// TwinCAT 3 PLC project ItemSimulator
// ProgramVersion: 3.1.4024.0
// libraries:
//   IO-Link Base, * (IO-Link)
//   SICK_IOL_Color, * (SICK AG)
//   Tc2_ModbusRTU, * (Beckhoff Automation GmbH)
//   Tc2_Standard, * (Beckhoff Automation GmbH)
//   Tc2_System, * (Beckhoff Automation GmbH)
//   Tc2_SystemCX, * (Beckhoff Automation GmbH)
//   Tc2_TcpIp, * (Beckhoff Automation GmbH)
//   Tc2_Utilities, * (Beckhoff Automation GmbH)
//   Tc3_Module, * (Beckhoff Automation GmbH)
//   TcUnit, * (www.tcunit.org)
//   VisuDialogs, * (System)
//   VisuSymbols,3.5.10.0,System
// project tree:
//   DUTs/ItemSimulator/ E_ItemGenerator.TcDUT, ST_ItemSimulator_HMI_CMD.TcDUT, ST_ItemSimulator_HMI_Status.TcDUT, ST_ItemSimulator_IO.TcDUT, ST_ItemGenerator.TcDUT
//   DUTs/TCP/ ST_TCPConnection.TcDUT, ST_TCPConnection_HMI_CMD.TcDUT, ST_TCPConnection_HMI_Status.TcDUT, ST_TCPConnection_IO.TcDUT
//   DUTs/TimeStamp/ ST_Timestamp_HMI_CMD.TcDUT, ST_Timestamp_HMI_Status.TcDUT, ST_Timestamp_IO.TcDUT
//   / GlobalTextList.TcGTLO, PlcTask.TcTTO, TCPTask.TcTTO, Visualization Manager.TcVMO (not stored)
//   GVLs/ GVL_Constant.TcGVL, GVL_HMI.TcGVL, GVL_IO.TcGVL
//   POUs/00_BuildingBlocks/ByteFunc/ FUN_GetHighByte.TcPOU, FUN_GetLowByte.TcPOU
//   POUs/00_BuildingBlocks/Calculation/ FB_FirstOrderLowPass.TcPOU, FUN_AngleCalculate.TcPOU, FUN_AngleChange.TcPOU, FUN_CartesianToPolar.TcPOU, FUN_Interpolation.TcPOU, FUN_LookUpTable.TcPOU, FUN_MinMaxSumAvg_6Reals.TcPOU, FUN_PolarToCartesian.TcPOU, FUN_Saturation.TcPOU, FUN_SaturationPointer.TcPOU, FUN_SaturationPointer_Int.TcPOU, FUN_SaturationPointer_UInt.TcPOU, FUN_Saturation_Int.TcPOU, FUN_Scale.TcPOU, ST_Coordinate.TcDUT
//   POUs/00_BuildingBlocks/Control/ FB_AliveCheck.TcPOU, FB_ClockPuls.TcPOU, FB_ClockPulsDetailed.TcPOU (not stored), FB_ClockPulsNumber.TcPOU, FB_EventHold.TcPOU, FB_FormatStringExtended.TcPOU, FB_Queue.TcPOU, FB_RampLimiter.TcPOU, FB_RangeSupervision.TcPOU, FB_SignalDead.TcPOU, FB_SteadyValue.TcPOU, FUN_InPos.TcPOU, FUN_InsideHysteresis.TcPOU, FUN_InsideHysteresis180pm.TcPOU, FUN_InsideHysteresis360.TcPOU, FUN_RangeInside.TcPOU, FUN_RangeOutside.TcPOU, FUN_GetHighLowValue.TcPOU
//   POUs/00_BuildingBlocks/Convert/ FUN_ConvFourByteToInt32.TcPOU, FUN_ConvFourByteToReal32.TcPOU, FUN_ConvFourByteToUdint32.TcPOU, FUN_ConvReal32ToFourByte.TcPOU, FUN_ConvTwoByteToInt16.TcPOU, FUN_ConvOneByteToUint8.TcPOU, FUN_ConvTwoByteToUInt16.TcPOU, U_Convert_INT16.TcDUT, U_Convert_UINT8.TcDUT, U_Convert_INT32.TcDUT, U_Convert_REAL32.TcDUT, U_Convert_UDINT32.TcDUT, U_Convert_UINT16.TcDUT, U_Convert_USINT.TcDUT
//   POUs/00_BuildingBlocks/EtherCAT/ FB_EK1101_Check.TcPOU, FB_HardwareCheck.TcPOU
//   POUs/00_BuildingBlocks/File/DUTs/ E_FileHandler_State.TcDUT
//   POUs/00_BuildingBlocks/File/ FB_FileHandler.TcPOU
//   POUs/00_BuildingBlocks/Modbus/DUTs/ E_ModbusRtuMaster_State.TcDUT, E_Modbus_DataType.TcDUT, ST_ModbusRtuMaster_StateLogEntry.TcDUT, ST_Modbus_Parameter.TcDUT, ST_Modbus_Unit.TcDUT
//   POUs/00_BuildingBlocks/Modbus/ FB_ModbusRtuMaster.TcPOU, FB_ModbusRtuMaster_20220719_1144.TcPOU, PRG_ModbusTest.TcPOU
//   POUs/00_BuildingBlocks/PlcToPlcCom/DUTs/ ADS_ErrorCodes.TcTLO, E_PlcAdsReadStep.TcDUT, ST_ComTest.TcDUT, ST_PlcAdsReadHmi.TcDUT
//   POUs/00_BuildingBlocks/PlcToPlcCom/ FB_PlcAdsRead.TcPOU, PRG_PlcAdsRead_Example.TcPOU, VIZU_PlcAdsRead.TcVIS
//   POUs/00_BuildingBlocks/StringFunctions/ FB_SeperateFileAndPathName.TcPOU, FUN_AddValuleToString.TcPOU, FUN_GetDateWithoutSeperator.TcPOU, FUN_GetDateWithUnderscore.TcPOU, FUN_GetDate.TcPOU, FUN_GetTimestamp.TcPOU, FUN_GetTimestampWithMs.TcPOU, FUN_GetTime.TcPOU, FUN_RealToString.TcPOU, FUN_ReplaceDotWithComma.TcPOU, F_Replace.TcPOU
//   POUs/01_TestUnit/ TEST.TcPOU (not stored)
//   POUs/01_TestUnit/TimeStampRegistry/ FB_TimestampRegistryTest.TcPOU
//   POUs/CSV_File/ PRG_CSVRead.TcPOU, PRG_CSVWrite.TcPOU (not stored)
//   POUs/IO_Link_Master/ FB_ColourSensor.TcPOU, FB_CMS.TcPOU, PRG_IO_Link_Master.TcPOU
//   POUs/Item_Simulator/FBs/ FB_ItemGenerator.TcPOU, FB_ItemRegister.TcPOU
//   POUs/Item_Simulator/ PRG_Simulator.TcPOU (not stored)
//   POUs/ MAIN.TcPOU, TCPCom.TcPOU
//   POUs/TCP_IP_Client/FBs/ FB_ReadTCP.TcPOU, FB_WriteTCP.TcPOU
//   POUs/TCP_IP_Client/ PRG_TCPIP.TcPOU
//   POUs/Timestamp_Registry/FBs/ FB_ReadTime.TcPOU (not stored), FB_SystemTime.TcPOU (not stored)
//   POUs/Timestamp_Registry/ PRG_TimestampRegistry.TcPOU
//   VISUs/ ItemSimulator.TcVIS, TimeStampOnItems.TcVIS
// real-time tasks:
//   TASK PlcTask: cycle T#10ms, priority 20, ADS port 350
//   TASK TCPTask: cycle T#2ms, priority 1, ADS port 351
// I/O:
//   DEVICE Device 5 (EtherCAT), AmsNetId 169.254.58.74.6.1
//     Box 1 (ICE11-8IOL-G60L-V1D) [ICE11-8IOL-G60L-V1D]
//       modules: Module 1 (IOL_I_32byte), Module 2 (IOL_I_32byte), Module 3 (IOL_I_16byte), Module 4 (IOL_I_16byte), Module 5 (IOL_I_16byte), Module 6 (IOL_I_16byte), Module 7 (IOL_I_16byte), Module 8 (IOL_I_16byte), Module 9 (STD_IN_1bit_Ch.B), Module 10 (STD_IN_1bit_Ch.B), Module 11 (STD_IN_1bit_Ch.B), Module 12 (STD_IN_1bit_Ch.B), Module 13 (STD_IN_1bit_Ch.B), Module 14 (STD_IN_1bit_Ch.B), Module 15 (STD_IN_1bit_Ch.B), Module 16 (STD_IN_1bit_Ch.B), Module 17 (TxPDO DI/IOL status), Module 18 (TxPDO New Diag Messages flag), Module 19 (TxPDO Timestamp), Module 20 (RxPDO DO/IOL control)
// variable links:
//   ItemSimulator/ItemSimulator Instance <-> Device 5 (EtherCAT)/Box 1 (ICE11-8IOL-G60L-V1D)
//     PlcTask Inputs/PRG_IO_Link_Master.fbCMS.arrCMSData <-> Module 2 (IOL_I_32byte)/TxPDO/input byte 0
//     PlcTask Inputs/PRG_IO_Link_Master.fbCMS.arrCMSData @bit {8..152 step 8} <-> Module 2 (IOL_I_32byte)/TxPDO/input byte {1..19}  (19 links)
//     PlcTask Inputs/PRG_IO_Link_Master.fbColorSensor.arrColorSensorData <-> Module 1 (IOL_I_32byte)/TxPDO/input byte 0
//     PlcTask Inputs/PRG_IO_Link_Master.fbColorSensor.arrColorSensorData @bit {8..88 step 8} <-> Module 1 (IOL_I_32byte)/TxPDO/input byte {1..11}  (11 links)
//     PlcTask Inputs/PRG_IO_Link_Master.fbColorSensor.nChannelStatus <-> IO-Link Port Status/Status of IO-Link Port 1

CONFIGURATION ItemSimulator
    RESOURCE PLC ON TwinCAT3
        TASK PlcTask(INTERVAL := T#10ms, PRIORITY := 20);
        TASK TCPTask(INTERVAL := T#2ms, PRIORITY := 1);
        PROGRAM MAIN WITH PlcTask : MAIN;
        PROGRAM TCPCom WITH TCPTask : TCPCom;
    END_RESOURCE
END_CONFIGURATION

// ---- DUTs/ItemSimulator/E_ItemGenerator.TcDUT
{attribute 'qualified_only'}
{attribute 'strict'}
TYPE E_ItemGenerator :
(
	Idle 						:= 0,
	ItemGenerator1 				:= 1,
	ItemGenerator2 				:= 2,
	ItemGenerator3 				:= 3,
	ItemGenerator4 				:= 4,
	ItemGenerator5 				:= 5,
	ItemGenerator6 				:= 6,
	ItemGenerator7 				:= 7,
	ItemGenerator8 				:= 8,
	ItemGenerator9 				:= 9,
	ItemGenerator10 			:= 10,
	ItemGeneratorFromRegistry	:= 11
	
);
END_TYPE

// ---- DUTs/ItemSimulator/ST_ItemSimulator_HMI_CMD.TcDUT
TYPE ST_ItemSimulator_HMI_CMD :
STRUCT
	bResetRegistry				:BOOL;
	bStartGenerator				:BOOL;
	bStopGenerator				:BOOL;
END_STRUCT
END_TYPE

// ---- DUTs/ItemSimulator/ST_ItemSimulator_HMI_Status.TcDUT
TYPE ST_ItemSimulator_HMI_Status :
STRUCT
END_STRUCT
END_TYPE

// ---- DUTs/ItemSimulator/ST_ItemSimulator_IO.TcDUT
TYPE ST_ItemSimulator_IO :
STRUCT
	bSignalOut	AT %Q* 			:BOOL;
	bSignalIn	AT %I* 			:BOOL;
END_STRUCT
END_TYPE

// ---- DUTs/ItemSimulator/ST_ItemGenerator.TcDUT
TYPE ST_ItemGenerator :
STRUCT
	bEnableGenerator		:BOOL;
	nNumberOfPulses			:UINT;
	tTimeOnPulse			:TIME;
	tTimeOffPulse			:TIME;
	bOutput					:BOOL;
END_STRUCT
END_TYPE

// ---- DUTs/TCP/ST_TCPConnection.TcDUT
TYPE ST_TCPConnection :
STRUCT
	bSocketConnect		:BOOL;
	sRemoteHost			:STRING;
	nRemotePort			:UDINT;
	tTimeOut			:TIME;
	bReset				:BOOL;
END_STRUCT
END_TYPE

// ---- DUTs/TCP/ST_TCPConnection_HMI_CMD.TcDUT
TYPE ST_TCPConnection_HMI_CMD :
STRUCT
	bWriteSocketConnect		:BOOL;
	bReadSocketConnect		:BOOL;
	bResetRegistry			:BOOL;
END_STRUCT
END_TYPE

// ---- DUTs/TCP/ST_TCPConnection_HMI_Status.TcDUT
TYPE ST_TCPConnection_HMI_Status :
STRUCT
	bCameraReadSocketIsConnected	:BOOL;
	bHlzWriteSocketIsConnected		:BOOL;
	
	aEANRegistry					:ARRAY[0..GVL_Constant.ITEM_ARRAY_SIZE] OF T_MaxString;
END_STRUCT
END_TYPE

// ---- DUTs/TCP/ST_TCPConnection_IO.TcDUT
TYPE ST_TCPConnection_IO :
STRUCT
END_STRUCT
END_TYPE

// ---- DUTs/TimeStamp/ST_Timestamp_HMI_CMD.TcDUT
TYPE ST_Timestamp_HMI_CMD :
STRUCT
	bResetRegistry				:BOOL;
END_STRUCT
END_TYPE

// ---- DUTs/TimeStamp/ST_Timestamp_HMI_Status.TcDUT
TYPE ST_Timestamp_HMI_Status :
STRUCT
	//Delta time in ms from Digital sensor to camera TCP
	aDeltaTimeMS			:ARRAY[0..GVL_Constant.ITEM_ARRAY_SIZE] OF UDINT;
	//Digital input sensor
	aDigitalSensorTime		:ARRAY[0..ITEM_ARRAY_SIZE] OF STRING;
	//Camera TCP port
	aTCPPortCameraTime		:ARRAY[0..ITEM_ARRAY_SIZE] OF STRING;
END_STRUCT
END_TYPE

// ---- DUTs/TimeStamp/ST_Timestamp_IO.TcDUT
TYPE ST_Timestamp_IO :
STRUCT
	bCameraOutSignal	AT %Q* 	:BOOL;
END_STRUCT
END_TYPE

// ---- POUs/00_BuildingBlocks/Calculation/ST_Coordinate.TcDUT
TYPE ST_Coordinate:
STRUCT
	rPosX			:LREAL;				// [mm] X-axis, Coordinate
	rPosY			:LREAL;				// [mm] Y-axis, Coordinate
	rPosTheta		:LREAL;				// [deg] Z-axis, Angle
END_STRUCT
END_TYPE

// ---- POUs/00_BuildingBlocks/Convert/U_Convert_INT16.TcDUT
TYPE U_Convert_INT16 :
UNION
	nValue		:INT;
	arrByte		:ARRAY[1..2] OF BYTE;
END_UNION
END_TYPE

// ---- POUs/00_BuildingBlocks/Convert/U_Convert_UINT8.TcDUT
TYPE U_Convert_UINT8 :
UNION
	nValue		:UINT;
	nBYTE		:BYTE;
END_UNION
END_TYPE

// ---- POUs/00_BuildingBlocks/Convert/U_Convert_INT32.TcDUT
TYPE U_Convert_INT32 :
UNION
	nValue		:DINT;
	arrByte		:ARRAY[1..4] OF BYTE;
END_UNION
END_TYPE

// ---- POUs/00_BuildingBlocks/Convert/U_Convert_REAL32.TcDUT
TYPE U_Convert_REAL32 :
UNION
	fValue		:REAL;
	arrByte		:ARRAY[1..4] OF BYTE;
END_UNION
END_TYPE

// ---- POUs/00_BuildingBlocks/Convert/U_Convert_UDINT32.TcDUT
TYPE U_Convert_UDINT32 :
UNION
	nValue		:UDINT;
	arrByte		:ARRAY[1..4] OF BYTE;
END_UNION
END_TYPE

// ---- POUs/00_BuildingBlocks/Convert/U_Convert_UINT16.TcDUT
TYPE U_Convert_UINT16 :
UNION
	nValue		:UINT;
	arrByte		:ARRAY[1..2] OF BYTE;
END_UNION
END_TYPE

// ---- POUs/00_BuildingBlocks/Convert/U_Convert_USINT.TcDUT
TYPE U_Convert_USINT :
UNION
	nValue		:USINT;					// Unsigned short integer value representation of data
    byValue 	:BYTE;					// Byte value representation of data
	//arrBit		:ARRAY[0..7]OF bool;	   // Bit representation of data
END_UNION
END_TYPE

// ---- POUs/00_BuildingBlocks/File/DUTs/E_FileHandler_State.TcDUT
{attribute 'qualified_only'}
{attribute 'strict'}
TYPE E_FileHandler_State :
(
	eReset				:= 0,
	eIdle				:= 10,
	
	eOpenFilePre		:= 20,
	eOpenFilePeri		:= 30,
	
	eReadFilePre		:= 40,
	eReadFilePeri		:= 50,

	eWriteFilePre		:= 60,
	eWriteFileSetLine	:= 65,
	eWriteFilePeri		:= 70,
	
	eCloseFilePre		:= 80,
	eCloseFilePeri		:= 90,

	eProcessFile		:= 100,
	
	eCopyFilePre		:= 200,
	eCopyFilePeri		:= 210,
	
	eDelFilePre			:= 220,
	eDelFilePeri		:= 230,
	
	eErrEntry			:= 900,
	eErrOpen			:= 910,
	eErrRead			:= 920,
	eErrWrite			:= 930,
	eErrClose			:= 940,
	eErrCopy			:= 950,
	eErrDel				:= 960
);
END_TYPE

// ---- POUs/00_BuildingBlocks/Modbus/DUTs/E_ModbusRtuMaster_State.TcDUT
{attribute 'qualified_only'}
{attribute 'strict'}
TYPE E_ModbusRtuMaster_State :
(
	eReset,
	eIdle,
	eReadPre,
	eReadPost,
	eError
);
END_TYPE

// ---- POUs/00_BuildingBlocks/Modbus/DUTs/E_Modbus_DataType.TcDUT
{attribute 'qualified_only'}
{attribute 'strict'}
TYPE E_Modbus_DataType :
(
	eInt16	 := 1,
	eInt32	 := 2
);
END_TYPE

// ---- POUs/00_BuildingBlocks/Modbus/DUTs/ST_ModbusRtuMaster_StateLogEntry.TcDUT
TYPE ST_ModbusRtuMaster_StateLogEntry :
STRUCT
	eStep				:E_ModbusRtuMaster_State;		// State
	sTimeEntry			:STRING;						// Timestamp for state entry
	iSecCount			:UDINT;							// Active time in state 	
END_STRUCT
END_TYPE

// ---- POUs/00_BuildingBlocks/Modbus/DUTs/ST_Modbus_Parameter.TcDUT
TYPE ST_Modbus_Parameter :
STRUCT
	nMemAddr			:WORD;
	nQuantity			:WORD;
	fConvFactor			:REAL;
	aDataStorage		:ARRAY[1..4] OF BYTE;
	aDataValue			:REAL;
	eDataType			:E_Modbus_DataType;
END_STRUCT
END_TYPE

// ---- POUs/00_BuildingBlocks/Modbus/DUTs/ST_Modbus_Unit.TcDUT
TYPE ST_Modbus_Unit :
STRUCT
	nAddr		:BYTE;
	aParam		:ARRAY[1..4] OF ST_Modbus_Parameter;		
END_STRUCT
END_TYPE

// ---- POUs/00_BuildingBlocks/PlcToPlcCom/DUTs/E_PlcAdsReadStep.TcDUT
//********************************************************************************
// E_PlcAdsReadStep
// ------------------------------------------------------------------------------- 
//
//	V2.00.00, HHL
// Baseline HST V1.01 10/4-16 (Valla V2.36)
//********************************************************************************
TYPE E_PlcAdsReadStep :
(
	eReset 				:= 0,		// Init
	eGetSymbolInfo 		:= 1,		// Get symbol infos
	eGetRemoteInfo 		:= 2,		// Get info (Index-Group/Offset)
	eWaitRemoteInfo 	:= 3,		// Wait for remote info
	eGetInfoError 		:= 4,		// Get info failed
	eIdle 				:= 10,		// Idle
	eRead 				:= 11,		// Read data
	eWaitReadDone 		:= 12,		// Wait read finished
	eWaitBeforeNextRead := 13, 		// Wait before next read
	eReadError 			:= 99		// Read failed
);
END_TYPE

// ---- POUs/00_BuildingBlocks/PlcToPlcCom/DUTs/ST_ComTest.TcDUT
TYPE ST_ComTest :
STRUCT
	bBool : BOOL;
	iInt : INT;
END_STRUCT
END_TYPE

// ---- POUs/00_BuildingBlocks/PlcToPlcCom/DUTs/ST_PlcAdsReadHmi.TcDUT
//********************************************************************************
// ST_PlcAdsReadHmi
// ------------------------------------------------------------------------------- 
//
//	V2.00.00, HHL
// Baseline HST V1.01 10/4-16 (Valla V2.36)
//********************************************************************************
TYPE ST_PlcAdsReadHmi :
STRUCT
	sRemoteId 				:STRING; 			// Remote NetId
	sRemoteSymbol 			:STRING;			// Remote variable
	bC_Init 				:BOOL; 				// Init request
	bS_Enable 				:BOOL; 				// Enable
	bS_LinkOk 				:BOOL; 				// Link to remote plc is ok
	bS_Error 				:BOOL; 				// Error
	eS_Step 				:E_PlcAdsReadStep;	// Step
	eS_ErrorStep		 	:E_PlcAdsReadStep;	// Error step
	udiS_ErrorId 			:UDINT; 			// Error id (ads)
	udiS_ReadCount 			:UDINT;  			// No of reads
	udiS_ReadErrors 		:UDINT; 			// No of read errors
	udiS_ReadIntervalErrors :UDINT;				// Read interval error
END_STRUCT
END_TYPE

// ---- GVLs/GVL_Constant.TcGVL
VAR_GLOBAL CONSTANT
	MAX_CSV_ROWS 			: UDINT := 100;
	MAX_CSV_COLUMNS 		: UDINT := 5;
	MAX_CSV_FIELD_LENGTH	: UDINT := 100;
	ITEM_ARRAY_SIZE			: INT:=10000;
END_VAR

// ---- GVLs/GVL_HMI.TcGVL
{attribute 'qualified_only'}
VAR_GLOBAL
	
	//Commands
	stItemSimulatorCmd		:ST_ItemSimulator_HMI_CMD;
	stTCPConnectionCmd		:ST_TCPConnection_HMI_CMD;
	stTimestampCmd			:ST_Timestamp_HMI_CMD;
	
	
	//Status
	stItemSimulatorStatus	:ST_ItemSimulator_HMI_Status;
	stTCPConnectionStatus	:ST_TCPConnection_HMI_Status;
	stTimestampStatus		:ST_Timestamp_HMI_Status;
END_VAR

// ---- GVLs/GVL_IO.TcGVL
{attribute 'qualified_only'}
VAR_GLOBAL
	stItemSimulator		:ST_ItemSimulator_IO;
	stTCPConnection		:ST_TCPConnection_IO;
	stTimestamp			:ST_Timestamp_IO;
END_VAR

// ---- POUs/MAIN.TcPOU
PROGRAM MAIN
VAR
END_VAR


//PRG_CSVRead();
//PRG_CSVWrite();

//Call Programs
PRG_Simulator();
PRG_TimestampRegistry();

PRG_IO_Link_Master();

END_PROGRAM

// ---- POUs/Timestamp_Registry/PRG_TimestampRegistry.TcPOU
PROGRAM PRG_TimestampRegistry
VAR 
	bInit					:BOOL := TRUE;
	fbReadTime				:FB_ReadTime;	
END_VAR

//Init
IF bInit THEN	
	bInit := FALSE;
END_IF

//Call read time
A_ReadTime();
	
//Reset Commands
GVL_HMI.stTimestampCmd.bResetRegistry := FALSE;

ACTION A_ReadTime:
fbReadTime(
	bReset := GVL_HMI.stTimestampCmd.bResetRegistry,
	bSignalIn := GVL_IO.stItemSimulator.bSignalIn,
	aDeltaTimeMS => GVL_HMI.stTimestampStatus.aDeltaTimeMS,
	aDigitalSensorTime => GVL_HMI.stTimestampStatus.aDigitalSensorTime,
	aTCPPortCameraTime => GVL_HMI.stTimestampStatus.aTCPPortCameraTime);
END_ACTION

END_PROGRAM

// ---- POUs/IO_Link_Master/PRG_IO_Link_Master.TcPOU
PROGRAM PRG_IO_Link_Master
VAR
	fbColorSensor			:FB_ColourSensor;
	fbCMS					:FB_CMS;
	
	bQL1					:BOOL; // Background
	bQL2					:BOOL; // Blue
	bQL3					:BOOL; // Green	
	bQL4					:BOOL; // None
	nQL1					:UINT;
	nQL2					:UINT;
	nQL3					:UINT;
	nQL4					:UINT;
	nValue					:INT;
	
	bEnable					:BOOL;
	bClear					:BOOL;
	arrColors				:ARRAY[0..GVL_Constant.ITEM_ARRAY_SIZE] OF INT;
	nI						:INT;
END_VAR

fbColorSensor(
	bQL1=>bQL1, 
	bQL2=>bQL2, 
	bQL3=>bQL3, 
	bQL4=>bQL4,
	nQL1=>nQL1,
	nQL2=>nQL2,
	nQL3=>nQL3,
	nQL4=>nQL4);
	
	
fbCMS();

nValue := fbColorSensor.nHighQLx;
IF NOT bQL1 AND NOT bClear THEN
	FOR nI := 0 TO GVL_Constant.ITEM_ARRAY_SIZE DO
		arrColors[nI] := fbColorSensor.nHighQLx;
	END_FOR
	
END_IF


IF bClear THEN
	FOR nI := 0 TO GVL_Constant.ITEM_ARRAY_SIZE DO
		arrColors[nI] := 0;
	END_FOR
END_IF

END_PROGRAM

// ---- POUs/IO_Link_Master/FB_ColourSensor.TcPOU
FUNCTION_BLOCK FB_ColourSensor
VAR_INPUT
END_VAR
VAR_OUTPUT
	nQL1					:UINT;
	nQL2					:UINT;
	nQL3					:UINT;
	nQL4					:UINT;
	
	bQL1					:BOOL;
	bQL2					:BOOL;
	bQL3					:BOOL;
	bQL4					:BOOL;
	
	nHighQLx				:INT;
END_VAR
VAR
	arrColorSensorData		AT %I*: ARRAY[0..11] OF BYTE;
	nChannelStatus			AT %I*: USINT;	
	
	arrQint					:ARRAY[1..24] OF BOOL;
	
	
	QoRAlarm				:BOOL;
	PDInvalid				:BOOL;
END_VAR

///////  index 120 value 0  ///////

// CMV QLx
nQL1 := FUN_ConvTwoByteToUInt16(nValue1 := arrColorSensorData[7], nValue2 := arrColorSensorData[6]); // CMV QL1
nQL2 := FUN_ConvTwoByteToUInt16(nValue1 := arrColorSensorData[5], nValue2 := arrColorSensorData[4]); // CMV QL2 
nQL3 := FUN_ConvTwoByteToUInt16(nValue1 := arrColorSensorData[3], nValue2 := arrColorSensorData[2]); // CMV QL3	
nQL4 := FUN_ConvTwoByteToUInt16(nValue1 := arrColorSensorData[1], nValue2 := arrColorSensorData[0]); // CMV QL4

IF bQL1 THEN
	nHighQLx := 1;
ELSIF bQL2 THEN
	nHighQLx := 2;
ELSIF bQL3 THEN
	nHighQLx := 3;
ELSIF bQL4 THEN
	nHighQLx := 4;
END_IF


// Qint 1 - 8
arrQint[1] := arrColorSensorData[10].0; //Not adjusted
arrQint[2] := arrColorSensorData[10].1; //Not adjusted
arrQint[3] := arrColorSensorData[10].2; //Not adjusted
arrQint[4] := arrColorSensorData[10].3; //Not adjusted
arrQint[5] := arrColorSensorData[10].4; //Not adjusted
arrQint[6] := arrColorSensorData[10].5; //Not adjusted
arrQint[7] := arrColorSensorData[10].6; //Not adjusted
arrQint[8] := arrColorSensorData[10].7; //Not adjusted

// Qint 9 - 16
arrQint[9] := arrColorSensorData[9].0; //Not adjusted
arrQint[10] := arrColorSensorData[9].1; //Not adjusted
arrQint[11] := arrColorSensorData[9].2; //Not adjusted
arrQint[12] := arrColorSensorData[9].3; //Not adjusted
arrQint[13] := arrColorSensorData[9].4; //Not adjusted
arrQint[14] := arrColorSensorData[9].5; //Not adjusted
arrQint[15] := arrColorSensorData[9].6; //Not adjusted
arrQint[16] := arrColorSensorData[9].7; //Not adjusted

// Qint 17 - 24
arrQint[17] := arrColorSensorData[8].0; //Not adjusted
arrQint[18] := arrColorSensorData[8].1; //Not adjusted
arrQint[19] := arrColorSensorData[8].2; //Not adjusted
arrQint[20] := arrColorSensorData[8].3; //Not adjusted
arrQint[21] := arrColorSensorData[8].4; //Not adjusted
arrQint[22] := arrColorSensorData[8].5; //Not adjusted
arrQint[23] := arrColorSensorData[8].6; //Not adjusted
arrQint[24] := arrColorSensorData[8].7; //Not adjusted

//Alarms
QoRAlarm := arrColorSensorData[11].4;
PDInvalid := arrColorSensorData[11].5;

//Digital outputs
bQL1 := arrColorSensorData[11].0;
bQL2 := arrColorSensorData[11].1;
bQL3 := arrColorSensorData[11].2;
bQL4 := arrColorSensorData[11].3;

END_FUNCTION_BLOCK

// ---- POUs/00_BuildingBlocks/Convert/FUN_ConvTwoByteToUInt16.TcPOU
FUNCTION FUN_ConvTwoByteToUInt16 : UINT
VAR_INPUT
	nValue1		:BYTE;				// Input Byte no 1
	nValue2		:BYTE;				// Input Byte no 2
END_VAR
VAR
	uData		:U_Convert_UINT16;		// Data variable used for conversion
END_VAR


// Save input bytes in data union
uData.arrByte[1] := nValue1;
uData.arrByte[2] := nValue2;

// Return value
FUN_ConvTwoByteToUInt16 := uData.nValue;

END_FUNCTION

// ---- POUs/IO_Link_Master/FB_CMS.TcPOU
FUNCTION_BLOCK FB_CMS
VAR_INPUT
END_VAR
VAR_OUTPUT
	Impulse_X				:REAL;
	Impulse_Y				:REAL;
	Impulse_Z				:REAL;
	Temperature				:REAL;
END_VAR
VAR
	arrCMSData				AT %I*: ARRAY[0..19] OF BYTE;
	nChannelStatus			AT %I*: USINT;	
	
	AlarmTemperature		:BOOL;
	AlarmShock				:BOOL;
	AlarmRMS_PreMax			:BOOL;
	AlarmRMS_Max			:BOOL;
	
	ConfByte				:ARRAY[0..1] OF BYTE;
END_VAR


Impulse_X := FUN_ConvFourByteToReal32(nValue1 := arrCMSData[15], nValue2 := arrCMSData[14], nValue3 := arrCMSData[13], nValue4 := arrCMSData[12]); 
Impulse_Y := FUN_ConvFourByteToReal32(nValue1 := arrCMSData[11], nValue2 := arrCMSData[10], nValue3 := arrCMSData[9], nValue4 := arrCMSData[8]); 
Impulse_Z := FUN_ConvFourByteToReal32(nValue1 := arrCMSData[7], nValue2 := arrCMSData[6], nValue3 := arrCMSData[5], nValue4 := arrCMSData[4]); 
Temperature := FUN_ConvFourByteToReal32(nValue1 := arrCMSData[3], nValue2 := arrCMSData[2], nValue3 := arrCMSData[1], nValue4 := arrCMSData[0]); 



// Byte 18 - 19 is configureable byte. These can be set in SOPAS software.
ConfByte[0].0 := arrCMSData[18].0; // Deactivated
ConfByte[0].1 := arrCMSData[18].1; // Deactivated
ConfByte[0].2 := arrCMSData[18].2; // Deactivated
ConfByte[0].3 := arrCMSData[18].3; // Deactivated
ConfByte[0].4 := arrCMSData[18].4; // Deactivated
ConfByte[0].5 := arrCMSData[18].5; // Deactivated
ConfByte[0].6 := arrCMSData[18].6; // Deactivated
ConfByte[0].7 := arrCMSData[18].7; // Deactivated

ConfByte[1].0 := arrCMSData[19].0; // Deactivated
ConfByte[1].1 := arrCMSData[19].1; // Deactivated
ConfByte[1].2 := arrCMSData[19].2; // Deactivated
ConfByte[1].3 := arrCMSData[19].3; // Deactivated

AlarmTemperature := arrCMSData[19].4; 
AlarmShock := arrCMSData[19].5; 
AlarmRMS_PreMax := arrCMSData[19].6; 
AlarmRMS_Max := arrCMSData[19].7;

END_FUNCTION_BLOCK

// ---- POUs/00_BuildingBlocks/Convert/FUN_ConvFourByteToReal32.TcPOU
FUNCTION FUN_ConvFourByteToReal32 : REAL
VAR_INPUT
	nValue1		:BYTE;				// Input Byte no 1
	nValue2		:BYTE;				// Input Byte no 2
	nValue3		:BYTE;				// Input Byte no 3
	nValue4		:BYTE;				// Input Byte no 4
END_VAR
VAR
	uData		:U_Convert_REAL32;	// Data variable used for conversion
END_VAR


// Save input bytes in data union
uData.arrByte[1] := nValue1;
uData.arrByte[2] := nValue2;
uData.arrByte[3] := nValue3;
uData.arrByte[4] := nValue4;

// Return value
FUN_ConvFourByteToReal32 := uData.fValue;

END_FUNCTION

// ---- POUs/TCPCom.TcPOU
PROGRAM TCPCom
VAR
END_VAR

//Call programs
PRG_TCPIP();

END_PROGRAM

// ---- POUs/TCP_IP_Client/PRG_TCPIP.TcPOU
PROGRAM PRG_TCPIP 
VAR	
	bInit 						:BOOL := TRUE;
	bReset						:BOOL;
	
	stReadTCP					:ST_TCPConnection;
	fbReadFromCameraTCP			:FB_ReadTCP;
	bConnectToReadSocket		:BOOL;
	
	stWriteTCP					:ST_TCPConnection;
	fbWriteToHLZ				:FB_WriteTCP;
	bConnectToWriteSocket		:BOOL;
END_VAR

//Init
IF bInit THEN	
	bInit := FALSE;
END_IF


A_ReadFromCamera();
A_WriteToHlz();


//Reset Commands
GVL_HMI.stTCPConnectionCmd.bResetRegistry := FALSE;


IF GVL_HMI.stTCPConnectionCmd.bWriteSocketConnect THEN
	GVL_HMI.stTCPConnectionCmd.bReadSocketConnect := FALSE;
	
ELSIF GVL_HMI.stTCPConnectionCmd.bReadSocketConnect THEN
	GVL_HMI.stTCPConnectionCmd.bWriteSocketConnect := FALSE;
END_IF;

ACTION A_ReadFromCamera:
//Initialize Read TCP
stReadTCP.sRemoteHost := '10.12.5.10';
stReadTCP.nRemotePort := 51236;
stReadTCP.tTimeOut := T#45S;
stReadTCP.bSocketConnect := GVL_HMI.stTCPConnectionCmd.bReadSocketConnect;
stReadTCP.bReset := GVL_HMI.stTCPConnectionCmd.bResetRegistry;

//Call Read TCP
fbReadFromCameraTCP(
	stTCPConnection:=stReadTCP,
	aEANRegistry=>GVL_HMI.stTCPConnectionStatus.aEANRegistry,
	bIsConnected=>GVL_HMI.stTCPConnectionStatus.bCameraReadSocketIsConnected);
END_ACTION

ACTION A_WriteToHlz:
//Initialize Write TCP
stWriteTCP.sRemoteHost := '10.12.5.10';
stWriteTCP.nRemotePort := 51237;
stWriteTCP.tTimeOut := T#45S;
stWriteTCP.bSocketConnect := GVL_HMI.stTCPConnectionCmd.bWriteSocketConnect;
stWriteTCP.bReset := GVL_HMI.stTCPConnectionCmd.bResetRegistry;


//Call Write TCP
fbWriteToHLZ(
	aEANRegistry:=fbReadFromCameraTCP.aEANRegistry,
	stTCPConnection:=stWriteTCP,
	bIsConnected=>GVL_HMI.stTCPConnectionStatus.bHlzWriteSocketIsConnected);
END_ACTION

END_PROGRAM

// ---- POUs/TCP_IP_Client/FBs/FB_ReadTCP.TcPOU
FUNCTION_BLOCK FB_ReadTCP 
VAR_INPUT
	stTCPConnection		:ST_TCPConnection;
END_VAR
VAR_OUTPUT
	aEANRegistry		:ARRAY[0..GVL_Constant.ITEM_ARRAY_SIZE] OF T_MaxString;
	bIsConnected		:BOOL;
END_VAR
VAR_IN_OUT
END_VAR
VAR
	fbConnectSocket		:FB_SocketConnect;
	fbDisconnect		:FB_SocketClose;
	rConnectedSocket	:F_TRIG;
	tRefreshRead		:FB_ClockPulsDetailed;
	fbSocketRecive		:FB_SocketReceive;
	rReadComplete		:R_TRIG;
	aReadBytes			:ARRAY[0..1023] OF BYTE;
	sReadString			:T_MaxString;
	iRead				:UINT;
	i					:INT;

	bReadComplete		:BOOL;
	bResetEANRegistry	:BOOL;
	hSocket				:T_HSOCKET;
END_VAR


A_ConnectToReadSocket();

IF bIsConnected THEN
	A_ReadFromTCPSocket();
END_IF

ACTION A_ConnectToReadSocket:
IF stTCPConnection.bSocketConnect THEN

	//Connect read port
	fbConnectSocket(
		sRemoteHost:=stTCPConnection.sRemoteHost,
		nRemotePort:=stTCPConnection.nRemotePort, 
		bExecute:=TRUE,
		tTimeout:=stTCPConnection.tTimeOut,
		hSocket=>hSocket);
	ELSE
		//Disconnect read port
		fbConnectSocket(bExecute:=FALSE);
		fbDisconnect(hSocket:=hSocket);
		bIsConnected := FALSE;
END_IF

rConnectedSocket(CLK:=fbConnectSocket.bBusy);

IF rConnectedSocket.Q AND NOT fbConnectSocket.bError THEN
	bIsConnected := TRUE;
END_IF
END_ACTION

ACTION A_ReadFromTCPSocket:
IF bIsConnected THEN

	//Refresh read timer
	tRefreshRead(bEnable:=TRUE, tPulsLengthOn:=T#2MS, tPulsLengthOff:=T#2MS);
	
	fbSocketRecive(
		hSocket:=hSocket, 
		cbLen:=SIZEOF(aReadBytes),
		pDest:=ADR(aReadBytes),
		bExecute:=tRefreshRead.bPuls);
		
	rReadComplete(CLK:=fbSocketRecive.nRecBytes > 0);
	
	
	//If byte read, copy into string.
	IF rReadComplete.Q THEN
		MEMCPY(destAddr:=ADR(sReadString), srcAddr:=ADR(aReadBytes),n:=fbSocketRecive.nRecBytes);
		aEANRegistry[iRead] := sReadString;
		MEMSET(destAddr:=ADR(aReadBytes),fillByte:=0, n:=fbSocketRecive.nRecBytes);
		MEMSET(destAddr:=ADR(sReadString),fillByte:=0, n:=fbSocketRecive.nRecBytes);
		iRead:=iRead+1;
		bReadComplete:=TRUE;
	ELSE
		bReadComplete:=FALSE;
	END_IF
END_IF


//Reset registry of EAN strings
IF PRG_Simulator.bStartGenerator OR PRG_Simulator.bStopGenerator OR (PRG_Simulator.i > PRG_Simulator.nTimeCount) OR stTCPConnection.bReset THEN
	FOR i := 0 TO GVL_Constant.ITEM_ARRAY_SIZE DO 
		aEANRegistry[i] := '';
	END_FOR

	iRead := 0;
	MEMSET(destAddr:=ADR(aReadBytes),fillByte:=0, n:=fbSocketRecive.nRecBytes);
	MEMSET(destAddr:=ADR(sReadString),fillByte:=0, n:=fbSocketRecive.nRecBytes);	
	
	
	//Reset commands
	stTCPConnection.bReset :=FALSE;
END_IF
END_ACTION

END_FUNCTION_BLOCK

// ---- POUs/TCP_IP_Client/FBs/FB_WriteTCP.TcPOU
FUNCTION_BLOCK FB_WriteTCP 
VAR_INPUT
	stTCPConnection		:ST_TCPConnection;
	aEANRegistry		:ARRAY[0..GVL_Constant.ITEM_ARRAY_SIZE] OF T_MaxString;
END_VAR
VAR_OUTPUT
	bIsConnected		:BOOL;
END_VAR
VAR
	fbConnectSocket		:FB_SocketConnect;
	fbDisconnect		:FB_SocketClose;
	rConnectedSocket	:F_TRIG;
	fbSocketSend		:FB_SocketSend;
	rWriteComplete		:R_TRIG;
	aWriteBytes			:ARRAY[0..1023] OF BYTE;
	iWrite				:UINT;
	WriteSignal			:F_TRIG;
	nWriteLen			:UDINT;
	i					:INT;

	bWriteComplete		:BOOL;
	bResetEANRegistry	:BOOL;
	hSocket				:T_HSOCKET;
END_VAR


A_ConnectToWriteSocket();

IF bIsConnected THEN
	A_WriteToTCPSocket();
END_IF

ACTION A_ConnectToWriteSocket:
IF stTCPConnection.bSocketConnect THEN
	
	//Connect write port
	fbConnectSocket(
		sRemoteHost:=stTCPConnection.sRemoteHost,
		nRemotePort:=stTCPConnection.nRemotePort, 
		bExecute:=TRUE,
		tTimeout:=stTCPConnection.tTimeOut,
		hSocket=>hSocket);
	ELSE
		//Disconnect write port
		fbConnectSocket(bExecute:=FALSE);
		fbDisconnect(hSocket:=hSocket);
		bIsConnected := FALSE;
END_IF



rConnectedSocket(CLK:=fbConnectSocket.bBusy);

IF rConnectedSocket.Q AND NOT fbConnectSocket.bError THEN
	bIsConnected := TRUE;
END_IF
END_ACTION

ACTION A_WriteToTCPSocket:
IF bIsConnected THEN	
	//Falling edge of item generator
	WriteSignal(CLK:=GVL_IO.stItemSimulator.bSignalOut);
	
	IF WriteSignal.Q THEN
		//Get length of string written
		nWriteLen := INT_TO_UDINT(LEN(STR:=aEANRegistry[iWrite]));
	
		//Copy string into array of bytes
		MEMCPY(destAddr:=ADR(aWriteBytes),srcAddr:=ADR(aEANRegistry[iWrite]),n:=nWriteLen);
		iWrite := iWrite + 1;
	END_IF
		
	//Write byte array to TCP server
	fbSocketSend(
		hSocket:=hSocket, 
		cbLen:=nWriteLen,
		pSrc:=ADR(aWriteBytes),
		bExecute:=WriteSignal.Q AND PRG_Simulator.fbItemGenerator.stItemGenFromReg.bEnableGenerator);
END_IF;


//Reset registry of EAN strings
IF PRG_Simulator.bStartGenerator OR PRG_Simulator.bStopGenerator OR (PRG_Simulator.i > PRG_Simulator.nTimeCount) OR bResetEANRegistry THEN
	FOR i := 0 TO GVL_Constant.ITEM_ARRAY_SIZE DO 
		aEANRegistry[i] := '';
	END_FOR

	iWrite := 0;	
	
	//Reset Command
	bResetEANRegistry := FALSE;
END_IF
END_ACTION

END_FUNCTION_BLOCK

// ---- POUs/00_BuildingBlocks/ByteFunc/FUN_GetHighByte.TcPOU
FUNCTION FUN_GetHighByte : BYTE
VAR_INPUT
	wIn			:WORD;			
END_VAR
VAR
	byHigh		:BYTE;
END_VAR


// Get the high byte value from the word
byHigh.0 := wIn.8;
byHigh.1 := wIn.9;
byHigh.2 := wIn.10;
byHigh.3 := wIn.11;
byHigh.4 := wIn.12;
byHigh.5 := wIn.13;
byHigh.6 := wIn.14;
byHigh.7 := wIn.15;

// Return value
FUN_GetHighByte := byHigh;

END_FUNCTION

// ---- POUs/00_BuildingBlocks/ByteFunc/FUN_GetLowByte.TcPOU
FUNCTION FUN_GetLowByte : BYTE
VAR_INPUT
	wIn			:WORD;			
END_VAR
VAR
	byLow		:BYTE;
END_VAR


// Get the high byte value from the word
byLow.0 := wIn.0;
byLow.1 := wIn.1;
byLow.2 := wIn.2;
byLow.3 := wIn.3;
byLow.4 := wIn.4;
byLow.5 := wIn.5;
byLow.6 := wIn.6;
byLow.7 := wIn.7;

// Return value
FUN_GetLowByte := byLow;

END_FUNCTION

// ---- POUs/00_BuildingBlocks/Calculation/FB_FirstOrderLowPass.TcPOU
//********************************************************************************
// FB_FirstOrderLowPass.
// -------------------------------------------------------------------------------
// This FB implements a first order low pass filter after the equation:
// 					Y[n] = Alpha x Y[n-1]  +  Beta X[n]
// The FB must be called in every scan when used. Input values for frequency and
// cut-off frequency can be changed during filtration without reset of the filtered
// output value.
//
// Version:
//			- V1.00.00	HHL, 26/11-2019
//********************************************************************************
FUNCTION_BLOCK FB_FirstOrderLowPass
VAR_INPUT
	rSampleFrequency	:REAL;			// Sample time for algorithm in Hz
	rCutOffFrequency	:REAL;			// Cut off frequency for filter in Hz 	
	rXn					:REAL;			// Input value before filtration
	bReset				:BOOL;			// Filter memory is reset on a rising edge. Output is reset to zero
END_VAR

VAR_OUTPUT
	rYn					:REAL;			// Output value after filtration
END_VAR

VAR
	osReset				:R_TRIG;		// One shot for reset of filter
	rFrequencyRatio		:REAL;			// Frequency ration for determination of Beta value
	rAlpha				:REAL;			// Alpha value for first order filter
	rBeta				:REAL;			// Beta value for first order filter
	rSampleFrequencyOld	:REAL;			// Input setting from previous scan for sample time for algorithm in Hz
	rCutOffFrequencyOld	:REAL;			// Input setting from previous scan for cut off frequency for filter in Hz 
END_VAR

// Check if filter has been reset
osReset(CLK:= bReset, Q=> );

// Check if settings have chaged
IF (rSampleFrequency <> rSampleFrequencyOld) OR (rCutOffFrequency <> rCutOffFrequencyOld) OR osReset.Q THEN
	// Settings have changed => Calculate Alpha and Beta again
	rFrequencyRatio := rSampleFrequency/rCutOffFrequency;
	rBeta := LREAL_TO_REAL(1/(2*PI*rFrequencyRatio));
	rAlpha := 1 - rBeta;
	
	// Update "old" values
	rSampleFrequencyOld := rSampleFrequency;
	rCutOffFrequencyOld := rCutOffFrequency;
	
	// If reset was activated, then reset output value
	IF osReset.Q THEN
		rYn := 0;
	END_IF
END_IF

// Calculate filtered value
rYn := rAlpha*rYn + rBeta*rXn;

END_FUNCTION_BLOCK

// ---- POUs/00_BuildingBlocks/Calculation/FUN_AngleCalculate.TcPOU
//********************************************************************************
// FUN_AngleCalculate.
// -------------------------------------------------------------------------------
// This function calculates the angle between two coordinate points.
// Angle when moving from stCoor1 to stCoor2 (Exit angle for stCoor1, Entry angle for stCoor2) 
// The output angle is defined as plus/minus 180 degrees. 
//	
// Version:
//			- V1.00.00	HHL, 26/11-2019
//********************************************************************************
FUNCTION FUN_AngleCalculate : LREAL
VAR_IN_OUT
END_VAR
VAR_INPUT
	stCoor1			:ST_Coordinate;			// Coordinates from previous motion command line (If known)
	stCoor2			:ST_Coordinate;			// Coordinates from active line
END_VAR
VAR
	rTheta			:LREAL;					// [pm 180 deg] Angle when moving from stCoor1 to stCoor2 (Exit angle for stCoor1, Entry angle for stCoor2) 
	bError			:BOOL;					// True if error occured during determination of angle
	rX_Leg			:LREAL;					// Displacement in x-axis between x-pos from stCoor1 and stCoor2
	rY_Leg			:LREAL;					// Displacement in y-axis between y-pos from stCoor1 and stCoor2
END_VAR

// Angle (Theta) must be calculated from two positions. 
// Calculate the two "legs" formed by the triangle of postion from stCoor1 and stCoor2 
rX_Leg := stCoor2.rPosX - stCoor1.rPosX;
rY_Leg := stCoor2.rPosY - stCoor1.rPosY;

// Calculate angle "Theta"
IF rX_Leg = 0 OR rY_Leg = 0 THEN
	// Theta is a parallel line to either x-axis or y-axis
	IF rX_Leg = 0 AND rY_Leg > 0 THEN
		// Theta is parallel to positive direction on y-axis
		rTheta := 90.0;
	ELSIF rX_Leg = 0 AND rY_Leg < 0 THEN
		// Theta is parallel to negative direction on y-axis
		rTheta := -90.0;
	ELSIF rX_Leg > 0 AND rY_Leg = 0 THEN
		// Theta is parallel to positive direction on x-axis
		rTheta := 0.0;
	ELSIF rX_Leg < 0 AND rY_Leg = 0 THEN
		// Theta is parallel to negative direction on x-axis
		rTheta := 180.0;
	ELSIF rX_Leg = 0 AND rY_Leg = 0 THEN
		// Special case where both stCoor1 and stCoor2 have the same coordinates (Should not happen).
		bError := TRUE;
	END_IF	
ELSE
	// Calculate angle "Theta" from position in stCoor1 and stCoor2	 
	IF stCoor1.rPosX <= stCoor2.rPosX AND stCoor1.rPosY <= stCoor2.rPosY THEN
		// I. Quadrant	
		// Location of stCoor2 in regards to stCoor1 as center
		IF rX_Leg <> 0 THEN
			rTheta := RAD_TO_DEG(ATAN(rY_Leg/rX_Leg));
		ELSIF rX_Leg = 0 THEN
			IF rY_Leg > 0 THEN
				rTheta := 90.0;
			ELSIF rY_Leg = 0 THEN
				// Special case where both stCoor1 and stCoor2 have the same coordinates (Should not happen).
				bError := TRUE;
			END_IF
		END_IF
	ELSIF stCoor1.rPosX > stCoor2.rPosX AND stCoor1.rPosY <= stCoor2.rPosY THEN 	
		// II. Quadrant	
		// Location of stCoor2 in regards to stCoor1 as centers
		IF rY_Leg <> 0 THEN
			rTheta := RAD_TO_DEG(ATAN(rY_Leg/rX_Leg)) + 180;
		ELSIF rY_Leg = 0 THEN
			IF rX_Leg > 0 THEN
				rTheta := 0.0;
			ELSE
				rTheta := -180.0;
			END_IF
		END_IF
	ELSIF stCoor1.rPosX > stCoor2.rPosX AND stCoor1.rPosY > stCoor2.rPosY THEN 	
		// III. Quadrant	
		// Location of stCoor2 in regards to stCoor1 as center
		rTheta := -1*(180 - RAD_TO_DEG(ATAN(rY_Leg/rX_Leg)));
	ELSIF stCoor1.rPosX < stCoor2.rPosX AND stCoor1.rPosY > stCoor2.rPosY THEN 	
		// IV. Quadrant	
		// Location of stCoor2 in regards to stCoor1 as center
		rTheta := RAD_TO_DEG(ATAN(rY_Leg/rX_Leg));
	END_IF	
END_IF

// Return result
IF NOT bError THEN
	// No error => Return result.
	FUN_AngleCalculate := rTheta;
ELSE
	// Error => Return error value
	FUN_AngleCalculate := -999.0;
END_IF

END_FUNCTION

// ---- POUs/00_BuildingBlocks/Calculation/FUN_AngleChange.TcPOU
//********************************************************************************
// FUN_AngleChange.
// -------------------------------------------------------------------------------
// This function calculates the difference between to angles in degrees. Input and
// output values are all defined as plus/minus 180 degrees. 
//	
// Version:
//			- V1.00.00	HHL, 26/11-2019
//********************************************************************************
FUNCTION FUN_AngleChange : LREAL
VAR_INPUT
	rTheta1			:LREAL;			// [pm 180 deg] Theta angle from coordinate set 1
	rTheta2			:LREAL;			// [pm 180 deg] Theta angle from coordinate set 2
END_VAR
VAR
	rThetaChange	:LREAL;			// Change in angle between two points	
END_VAR

// Calculate change in theta angle
IF rTheta1 >= 0 AND rTheta2 >= 0 THEN
	// Both coordinates have a positive theta angle
	rThetaChange := rTheta2 - rTheta1;
ELSIF rTheta1 <= 0 AND rTheta2 <= 0 THEN
	// Both coordinates have a negative thata angle
	rThetaChange := rTheta2 - rTheta1;
ELSE
	// One coordinate set has a positive theta angle and the other has a negative
	IF rTheta1 >= 0 THEN
		// Coordinate set one has a positive coordinate set and coordinate 2 has a negative
		// First find angle when passing through 0 deg.
		rThetaChange := rTheta2 - rTheta1;
		IF ABS(rThetaChange) > 180 THEN
			// Angle is greather than 180 deg. Do not use angle that passes through 0 deg. 
			// Calculate the angle when passing through p/m 180 deg
			rThetaChange := 360 - ABS(rThetaChange);
		END_IF
	ELSE
		// Coordinate set one has a negative coordinate set and coordinate 2 has a positive
		// First find angle when passing through 0 deg.
		rThetaChange := rTheta2 - rTheta1;
		IF ABS(rThetaChange) > 180 THEN
			// Angle is greather than 180 deg. Do not use angle that passes through 0 deg. 
			// Calculate the angle when passing through p/m 180 deg
			rThetaChange := -1 * (360 - ABS(rThetaChange));
		END_IF
	END_IF
END_IF 

// Return result
FUN_AngleChange := rThetaChange;

END_FUNCTION

// ---- POUs/00_BuildingBlocks/Calculation/FUN_CartesianToPolar.TcPOU
//********************************************************************************
// FUN_Cartesian to polar.
// -------------------------------------------------------------------------------
// This function calculates the polar coordinates r and theta from
// the cartesian X and Y coordinates. 
//	
// Version:
//			- V1.01	HHL, 11/05-2022
//********************************************************************************
FUNCTION FUN_CartesianToPolar : LREAL
VAR_IN_OUT
END_VAR
VAR_INPUT
	fX				:REAL;			// X-axis coordinate
	fY				:REAL;			// Y-axis coordinate
END_VAR
VAR_OUTPUT
	fRadius			:REAL;			// Radius for polar coordinate
	fAngle			:REAL;			// [deg] Angle for polar coordinate 
END_VAR
VAR
	bError			:BOOL;			// True if error occured during determination of angle
END_VAR


// Calculate polar coordinates from cartesian coordinates
//-----------------------------------------

// Calculate radius
fRadius := LREAL_TO_REAL(SQRT((EXPT(fX,2) + EXPT(fY,2))));

// Calculate angle
IF fX <> 0 THEN 
	// Calculate angle 
	IF 0 <= fX AND 0 <= fY THEN
		// I. Quadrant	
		IF fX <> 0 THEN
			fAngle := LREAL_TO_REAL(RAD_TO_DEG(ATAN(fY/fX)));
		ELSIF fX = 0 THEN
			IF fY > 0 THEN
				fAngle := 90.0;
			ELSIF fY = 0 THEN
				// Special case where both fX and fY are zero.
				bError := TRUE;
			END_IF
		END_IF
	ELSIF 0 > fX AND 0 <= fY THEN 	
		// II. Quadrant	
		IF fY <> 0 THEN
			fAngle := LREAL_TO_REAL(RAD_TO_DEG(ATAN(fY/fX)) + 180);
		ELSIF fY = 0 THEN
			IF fX > 0 THEN
				fAngle := 0.0;
			ELSE
				fAngle := -180.0;
			END_IF
		END_IF
	ELSIF 0 > fX AND 0 > fY THEN 	
		// III. Quadrant	
		fAngle := -1*(180 - LREAL_TO_REAL(RAD_TO_DEG(ATAN(fY/fX))));
	ELSIF 0 < fX AND 0 > fY THEN 	
		// IV. Quadrant	
		fAngle := LREAL_TO_REAL(RAD_TO_DEG(ATAN(fY/fX)));
	END_IF	
ELSE
	// X-axis coordinate is zero 
	IF fY = 0 THEN
		fAngle  := 0.0;		
	ELSIF fY > 0 THEN
		fAngle  := 90.0;
	ELSE
 		fAngle  := -90.0;
	END_IF
END_IF

END_FUNCTION

// ---- POUs/00_BuildingBlocks/Calculation/FUN_Interpolation.TcPOU
///*****************************************************************************************
///            Simple interpolation function for two points (X1,X2) and (Y1,Y2)                
///*****************************************************************************************
FUNCTION FUN_Interpolation : REAL
VAR_INPUT
	rInputValue: REAL;
	rX1: REAL;
	rY1: REAL;
	rX2: REAL;
	rY2: REAL;
END_VAR
VAR
	rSlope: REAL;
END_VAR

(*The slope between the two points (X1,Y1) and (X2,Y2) is calculated*)
IF (rX2-rX1) <> 0 THEN
	rSlope := (rY2-rY1)/(rX2-rX1);
ELSE
	rSlope := 0;
END_IF

(*The output value is calculated from the slope and input*)
FUN_Interpolation := rY1 + rSlope*(rInputValue-rX1);

END_FUNCTION

// ---- POUs/00_BuildingBlocks/Calculation/FUN_LookUpTable.TcPOU
FUNCTION FUN_LookUpTable : REAL
VAR_INPUT
	iNumberOfPoints			:INT;						(* Specifies the number of points in the loopup table. Min 2 and max 10 *)
	rInput					:REAL;						(* Input value to look up table *)
	arrAxisX				:ARRAY[1..10] OF REAL;		(* Definition of lookup table, points on x-axis, Min 2 and max 10 *)
	arrAxisY				:ARRAY[1..10] OF REAL;		(* Definition of lookup table, points on y-axis, Min 2 and max 10 *)
END_VAR
VAR
	rOutput					:REAL;						(* Look up table output value *)
	bError					:BOOL;						(* TRUE if number of input points are nonvalid *)
	bMakeLookUp				:BOOL;						(* FALSE if input value is outside min and max values on x-axis. Output is saturated *)
	bIndexHighFound			:BOOL;						(* TRUE when the high index is found *)
	iIndexHigh				:INT;						(* Holds the high index value on the lookup table for  the input value *)
	iIndexLow				:INT;						(* Holds the low index value on the lookup table for the input value*)
	iIndex					:INT;						(* index counter *)
END_VAR


(* Check if number of points are valid *)
IF iNumberOfPoints < 2 OR iNumberOfPoints > 10 THEN
	bError := TRUE;
ELSE
	bError := FALSE;
END_IF

(* Check input value, is it within the x-axis min and max points. If yes then make calculation,
    if no then saturate to min and max values											 *)
IF rInput >= arrAxisX[iNumberOfPoints] THEN
	rOutput := arrAxisY[iNumberOfPoints];
ELSIF rInput <= arrAxisX[1] THEN
	rOutput := arrAxisY[1];
ELSE
	bMakeLookUp := TRUE;
END_IF


(* Find high and low index for input value *)
IF bMakeLookUp AND NOT bError THEN

	(* While loop findes high index *)
	iIndex := 1;
	WHILE NOT bIndexHighFound AND iIndex <= iNumberOfPoints DO
		IF rInput <= arrAxisX[iIndex] THEN
			iIndexHigh := iIndex;
			bIndexHighFound := TRUE;
		END_IF
		iIndex := iIndex +1;
	END_WHILE
	iIndexLow := iIndexHigh - 1;

	(* Make interpolation between high and low value *)
	rOutput := FUN_Interpolation(rInput, arrAxisX[iIndexLow], arrAxisY[iIndexLow], arrAxisX[iIndexHigh], arrAxisY[iIndexHigh]);

	(* Clean up before next run *)
	bIndexHighFound := FALSE;
	bMakeLookUp := FALSE;
END_IF

FUN_LookUpTable := rOutput;

END_FUNCTION

// ---- POUs/00_BuildingBlocks/Calculation/FUN_MinMaxSumAvg_6Reals.TcPOU
//Last update: 2022-07-08/BJST
FUNCTION FUN_MinMaxSumAvg_6Reals : REAL	//Return average value	
VAR_INPUT
	fVal_1	:REAL;
	fVal_2	:REAL;
	fVal_3	:REAL;
	fVal_4	:REAL;
	fVal_5	:REAL;
	fVal_6	:REAL;
END_VAR
VAR
	afVal	:ARRAY [1..6] OF REAL;
END_VAR
VAR_OUTPUT
	n		:INT;
	fMin	:REAL;
	fMax	:REAL;
	fSum	:REAL;
	fAvg	:REAL;
END_VAR

//Read inputs

//Read inputs
afVal[1] := fVal_1;
afVal[2] := fVal_2;
afVal[3] := fVal_3;
afVal[4] := fVal_4;
afVal[5] := fVal_5;
afVal[6] := fVal_6;

//Initialize
fSum := fAvg := 0;
fMin := fMax := afVal[1];

//Calculate
FOR n:=1 TO 6 DO
	fSum := fSum + afVal[n];
	IF fMin > afVal[n] THEN	fMin := afVal[n];	END_IF
	IF fMax < afVal[n] THEN	fMax := afVal[n];	END_IF
END_FOR

fAvg := fSum/6;

END_FUNCTION

// ---- POUs/00_BuildingBlocks/Calculation/FUN_PolarToCartesian.TcPOU
//********************************************************************************
// FUN_PolarToCartesian.
// -------------------------------------------------------------------------------
// This function calculates the cartesian X and Y coordinates from the 
// polar coordinates r and theta.
//	
// Version:
//			- V1.00.00	HHL, 01/04-2021
//********************************************************************************
FUNCTION FUN_PolarToCartesian : BOOL
VAR_IN_OUT
END_VAR
VAR_INPUT
	fRadius			:REAL;			// Radius for polar coordinate
	fAngle			:REAL;			// [deg] Angle for polar coordinate 
END_VAR
VAR_OUTPUT
	fX				:REAL;			// X-axis coordinate
	fY				:REAL;			// Y-axis coordinate	
END_VAR


// Calculate cartesian coordinates from polar coordinates
fX := LREAL_TO_REAL(fRadius * COS(DEG_TO_RAD(fAngle)));
fY := LREAL_TO_REAL(fRadius * SIN(DEG_TO_RAD(fAngle)));

END_FUNCTION

// ---- POUs/00_BuildingBlocks/Calculation/FUN_Saturation.TcPOU
/// Saturation function. Limits the input to a minimum and maximum value
FUNCTION FUN_Saturation : REAL
VAR_INPUT
	rInputValue		:REAL;				// Input value before saturation				
	rOutputMin		:REAL;				// Saturation min value
	rOutputMax		:REAL;				// Saturation max value
END_VAR
VAR
	rOutputValue	:REAL;				// Output value after saturation
END_VAR

IF rInputValue > rOutputMin THEN
	IF rInputValue < rOutputMax THEN
		rOutputValue := rInputValue;
	ELSE
		rOutputValue := rOutputMax;
	END_IF
ELSE
	rOutputValue := rOutputMin;
END_IF

FUN_Saturation := rOutputValue;

END_FUNCTION

// ---- POUs/00_BuildingBlocks/Calculation/FUN_SaturationPointer.TcPOU
/// Saturation. Limits the value to a minimum and maximum value
FUNCTION FUN_SaturationPointer : REAL
VAR_INPUT
	pValue			:POINTER TO REAL;	// Value				
	fMin			:REAL;				// Saturation min value
	fMax			:REAL;				// Saturation max value
END_VAR
VAR_OUTPUT
	bSaturation		:BOOL;
END_VAR

bSaturation := FALSE;
IF pValue^ < fMin THEN
	pValue^ := fMin;
	bSaturation := TRUE;
ELSIF pValue^ > fMax THEN
	pValue^ := fMax;
	bSaturation := TRUE;
END_IF

END_FUNCTION

// ---- POUs/00_BuildingBlocks/Calculation/FUN_SaturationPointer_Int.TcPOU
/// Saturation. Limits the value to a minimum and maximum value
FUNCTION FUN_SaturationPointer_Int : REAL
VAR_INPUT
	pValue			:POINTER TO INT;	// Value				
	fMin			:REAL;				// Saturation min value
	fMax			:REAL;				// Saturation max value
END_VAR
VAR_OUTPUT
	bSaturation		:BOOL;
END_VAR

bSaturation := FALSE;
IF INT_TO_REAL(pValue^) < fMin THEN
	pValue^ := REAL_TO_INT(fMin);
	bSaturation := TRUE;
ELSIF INT_TO_REAL(pValue^) > fMax THEN
	pValue^ := REAL_TO_INT(fMax);
	bSaturation := TRUE;
END_IF

END_FUNCTION

// ---- POUs/00_BuildingBlocks/Calculation/FUN_SaturationPointer_UInt.TcPOU
/// Saturation. Limits the value to a minimum and maximum value
FUNCTION FUN_SaturationPointer_UInt : REAL
VAR_INPUT
	pValue			:POINTER TO UINT;	// Value				
	fMin			:REAL;				// Saturation min value
	fMax			:REAL;				// Saturation max value
END_VAR
VAR_OUTPUT
	bSaturation		:BOOL;
END_VAR

bSaturation := FALSE;
IF UINT_TO_REAL(pValue^) < fMin THEN
	pValue^ := REAL_TO_UINT(fMin);
	bSaturation := TRUE;
ELSIF UINT_TO_REAL(pValue^) > fMax THEN
	pValue^ := REAL_TO_UINT(fMax);
	bSaturation := TRUE;
END_IF

END_FUNCTION

// ---- POUs/00_BuildingBlocks/Calculation/FUN_Saturation_Int.TcPOU
/// Saturation function. Limits the input to a minimum and maximum value
FUNCTION FUN_Saturation_Int : REAL
VAR_INPUT
	/// Input value before saturation	
	InputValue: REAL;
	/// Saturation min value			
	OutputMin: REAL;
	/// Saturation max value			
	OutputMax: REAL;
END_VAR
VAR
	OutputValue: REAL;
END_VAR

IF InputValue > OutputMin THEN
	IF InputValue < OutputMax THEN
		OutputValue := InputValue;
	ELSE
		OutputValue := OutputMax;
	END_IF
ELSE
	OutputValue := OutputMin;
END_IF

FUN_Saturation := OutputValue;

END_FUNCTION

// ---- POUs/00_BuildingBlocks/Calculation/FUN_Scale.TcPOU
///**********************************************************************************
///    Scales input value based on interpolation between input and output
///      min and max values                                                                                              
///**********************************************************************************
FUNCTION FUN_Scale : REAL
VAR_INPUT
	///  The input that is to be scaled	 
	fInputValue: REAL;
	/// The minimum allowable input	 
	fInputMin: REAL;
	/// The maximum allowable input	 
	fInputMax: REAL;
	/// The minimum allowable ouput	 
	fOutputMin: REAL;
	/// The maximum allowable ouput	 
	fOutputMax: REAL;
END_VAR
VAR
	fTemp: REAL;
END_VAR

fTemp := FUN_Interpolation(fInputValue, fInputMin, fOutputMin, fInputMax, fOutputMax);
FUN_Scale := FUN_Saturation(fTemp, fOutputMin, fOutputMax);

END_FUNCTION

// ---- POUs/00_BuildingBlocks/Control/FB_AliveCheck.TcPOU
//********************************************************************************
// FB_AliveCheck
// -------------------------------------------------------------------------------
// This function block is used to check if an alive signal is present. An alive signal
// is assumed to be a clock puls. An alarm is set if the clock puls is missing or frozen. 
// 
// Version:
//			- V1.00.00	HHL, 08/08-2019
//********************************************************************************
FUNCTION_BLOCK FB_AliveCheck
VAR_INPUT
	bEnable				:BOOL;			// When true alive check is performed
	bSignal				:BOOL;			// Alive signal
	tStartDelay			:TIME;			// Time from boot to activation of check 
	tTimeout			:TIME;			// Time untill timeout occurs when alive signal is lost
	bReset				:BOOL;			// Reset of alarm
END_VAR
VAR_OUTPUT
	bAlarm				:BOOL;			// True if alive signal was lost			
END_VAR
VAR
	tonStartUpDelay		:TON;			// Delay from boot to start of check
	bAlive				:BOOL;			// Set true when alive signal is received
	osAlive				:R_TRIG;		// One shot for rising edge on alive bit
	tonAliveTO			:TON;			// Timeout for missing alive signal
END_VAR


// Initialize alive signal to false
bAlive := FALSE;
// Check for rising edge on input sinal (clock puls signal from external device)
osAlive(CLK:= bSignal, Q=> );
IF osAlive.Q THEN
	// Alive puls is registered, set alive flag => Reset timer for alarm
	bAlive := TRUE;
END_IF

// Update startup timer (boot) 
tonStartUpDelay(IN:= TRUE, PT:= tStartDelay, Q=> , ET=> );

// Check for timeout and set alam signal
tonAliveTO(IN:= bEnable AND NOT bAlive AND tonStartUpDelay.Q, PT:= tTimeout, Q=> , ET=> );
IF tonAliveTO.Q THEN
	// Timeout, Alive signal is missing => set alarm
	bAlarm := TRUE;
ELSE 
	// Auto reset
	bAlarm := FALSE;
END_IF

IF ((NOT bEnable AND bAlarm) OR bReset) THEN
	// Reset 
	bAlarm := FALSE;
END_IF

END_FUNCTION_BLOCK

// ---- POUs/00_BuildingBlocks/Control/FB_ClockPuls.TcPOU
// This vunction block creates a clock puls. The function block is useful when
// somthing needs to be trigged with a fixed frequency. Note that the variable
// tPulsLength defines the time between two rising edges in the clock puls
FUNCTION_BLOCK FB_ClockPuls
VAR_INPUT
	bEnable				:BOOL;		// When TRUE a clock puls is generated. If set FALSE the bPuls output is always FALSE
	tPulsLength			:TIME;		// Time for one complete clock puls. 											      
END_VAR

VAR_OUTPUT
	bPuls				:BOOL;		// Clock Puls
END_VAR

VAR
	fbTimer1			:TON;		// Internal timer
	fbTimer2			:TON;		// Internal timer
	tHalfPuls			:TIME;
	bTimerOut			:BOOL;
END_VAR

// Calculate the time for half a clock puls
tHalfPuls := tPulsLength/2;

// Generate clock puls
IF bEnable THEN
	fbTimer1(IN:= NOT fbTimer2.Q , PT:= tHalfPuls, Q=>bTimerOut , ET=> );
	fbTimer2(IN:= fbTimer1.Q, PT:= tHalfPuls, Q=> , ET=> );
	// Start with postive edge when enabled
	bPuls := NOT bTimerOut;	
ELSE
	fbTimer1(IN:=FALSE);
	fbTimer2(IN:=FALSE);
	bPuls := FALSE;
END_IF

END_FUNCTION_BLOCK

// ---- POUs/00_BuildingBlocks/Control/FB_ClockPulsNumber.TcPOU
FUNCTION_BLOCK FB_ClockPulsNumber
VAR_INPUT
	bTrig				:BOOL;					// On a rising edge, uiNo of puls are generated
	bStop				:BOOL;					// Stop and reset pulses
	uiNo				:UINT;					// Number of pulses to be generated when bTrig is set high
	tPulsLengthOn 		:TIME;
	tPulsLengthOff 		:TIME;
END_VAR
VAR_OUTPUT
	bPuls				:BOOL;					// Output puls
END_VAR
VAR
	osTrig				:R_TRIG;				// One shot trigger for start of pulses
	osPuls				:R_TRIG;				// One shot trigger for output puls
	uiCount				:UINT;					// Reset puls count
	fbStart				:SR;					// Set/Reset for reset to main zone.
	fbClockPulsDetailed :FB_ClockPulsDetailed;
END_VAR



// Wait	for trig signal
osTrig(CLK:= bTrig, Q=> );

// Set start signal
fbStart(SET1:= osTrig.Q, RESET:= (uiCount > uiNo) OR bStop, Q1=> );

// Reset start signal
IF fbStart.RESET THEN
	uiCount := 0;
END_IF

// Generate clock puls
fbClockPulsDetailed(bEnable:= fbStart.Q1 AND NOT bStop, tPulsLengthOn := tPulsLengthOn, tPulsLengthOff:= tPulsLengthOff, bPuls=>);

// Count number of output pulses
osPuls(CLK:= fbClockPulsDetailed.bPuls, Q=> );
IF osPuls.Q THEN
	uiCount := uiCount + 1;
END_IF

// Set output puls
IF uiCount <= uiNo THEN
	bPuls := fbClockPulsDetailed.bPuls;
ELSE
	bPuls := FALSE;
END_IF

END_FUNCTION_BLOCK

// ---- POUs/00_BuildingBlocks/Control/FB_EventHold.TcPOU
FUNCTION_BLOCK FB_EventHold
VAR_INPUT
	bEvent		:BOOL;
END_VAR
VAR_OUTPUT
	bEventHold	:BOOL;
END_VAR
VAR
	osTrig		:R_TRIG;
	srEvent		:SR;
	tonHold		:TON;
END_VAR


// One shot trigger for event
osTrig(CLK:= bEvent, Q=> );

// Remember that event has been activated, and hold it untill reset
srEvent(
	SET1:= osTrig.Q, 
	RESET:= tonHold.Q, Q1=> );

// Reset after xx MS
tonHold(IN:= srEvent.Q1, PT:= T#500MS, Q=> , ET=> );

// Set Event Hold
bEventHold := srEvent.Q1;

END_FUNCTION_BLOCK

// ---- POUs/00_BuildingBlocks/Control/FB_FormatStringExtended.TcPOU
FUNCTION_BLOCK FB_FormatStringExtended
VAR_INPUT
	pFormatString : POINTER TO STRING;
    arg1      : T_Arg;
    arg2      : T_Arg;
    arg3      : T_Arg;
    arg4      : T_Arg;
    arg5      : T_Arg;
    arg6      : T_Arg;
    arg7      : T_Arg;
    arg8      : T_Arg;
    arg9      : T_Arg;
    arg10     : T_Arg;
	arg11      : T_Arg;
    arg12      : T_Arg;
    arg13      : T_Arg;
    arg14      : T_Arg;
    arg15      : T_Arg;
    arg16      : T_Arg;
    arg17      : T_Arg;
    arg18      : T_Arg;
    arg19      : T_Arg;
    arg20     : T_Arg;
	pDstString    : POINTER TO STRING;
    nDstSize      : UDINT;
END_VAR
VAR_OUTPUT
	bError : BOOL;
    nErrId : UDINT;
END_VAR
VAR
END_VAR

END_FUNCTION_BLOCK

// ---- POUs/00_BuildingBlocks/Control/FB_Queue.TcPOU
FUNCTION_BLOCK FB_Queue
VAR_INPUT
END_VAR
VAR_OUTPUT
	bFull	 				:BOOL := FALSE;					// True if queue is full
	iNoOfEntries			:UINT := 0;						// Number of entries in the queue
	iNoOfFree				:UINT := cQueueSize; // Number of free entries
END_VAR
VAR
	iInputIndex 			:UINT := 1;						// Points to next input entry in queue
	iOutputIndex	 		:UINT := 1;						// Points to next output entry in queue
 	arrQueue	 			:ARRAY[1..cQueueSize] OF INT;	// Queue
	bError					:BOOL;							// True if error occurs
END_VAR
VAR CONSTANT
	cQueueSize				:UINT := 100;				
END_VAR

METHOD M_Flush : BOOL
VAR_INPUT
END_VAR
VAR
	iEntryEmpty		:INT;			// Entry with zero content
	iForIndex		:INT;			// Index used in for-loops	
END_VAR

// Flush Queue. All entries are deleted. Index's and counters are reset.
//----------------------------------------------------------------------

// Initialize empty entry
iEntryEmpty := 0;

// Reset all entries in queue
FOR iForIndex := 1 TO UINT_TO_INT(cQueueSize) BY 1 DO
	arrQueue[iForIndex] := iEntryEmpty;
END_FOR

// Reset index's and counters
iInputIndex 	:= 1;
iOutputIndex	:= 1;
iNoOfEntries	:= 0;
iNoOfFree		:= cQueueSize;
END_METHOD

METHOD M_GetEntry : BOOL
VAR_OUTPUT
	iEntry 				:INT;			// Value for found entry in queue 
	bNewEntry			:BOOL;			// True if new entry was foud in queue, False if queue is empty
END_VAR

// Check if there are any events in queue
IF(iInputIndex <> iOutputIndex ) THEN							
	// Min one event in queue, get next event
	iEntry := arrQueue[iOutputIndex];		
	bNewEntry := TRUE;
											
	// Update output index	
  	IF(iOutputIndex > (cQueueSize-1)) THEN 									
  		iOutputIndex := 1;
  	ELSE
		iOutputIndex := iOutputIndex + 1;
	END_IF
	
	// Update the entry counter
	iNoOfEntries := iNoOfEntries - 1;
	
	// Reset full flag if it was set
	bFull := FALSE; 
ELSE
	// No events in queue
	bNewEntry := FALSE;
	iNoOfEntries := 0;
END_IF;

// Update count for number of free entires
iNoOfFree := cQueueSize - iNoOfEntries;
END_METHOD

METHOD M_GetFullStatus : BOOL
VAR_INPUT
END_VAR
// Returns true if queue is full

// Initialize to false
M_GetFullStatus := FALSE;

// Update signal
IF((iInputIndex+1) > cQueueSize) THEN
	// Input index will loop around at next entry. Make sure that output index is not occuping this place.
	IF iOutputIndex = 0 THEN
		M_GetFullStatus := TRUE;
	END_IF
ELSIF ((iInputIndex + 1) = iOutputIndex) THEN
	// Output is occuping next entry. Queue full 
	M_GetFullStatus := TRUE;
END_IF

// Check entry counter	
IF iNoOfEntries >= cQueueSize THEN
	M_GetFullStatus := TRUE;
END_IF
END_METHOD

METHOD M_PutEntry : BOOL
VAR_INPUT
	iEntry	 		:INT;			// Value to be stored in queue
END_VAR

// Update Full flag
IF iNoOfEntries >= cQueueSize THEN
	bFull := TRUE;
ELSE
	bFull := FALSE;
END_IF


// Put entry into queue unless it is full
IF NOT bFull THEN
	arrQueue[iInputIndex] := iEntry;
	iNoOfEntries := iNoOfEntries + 1;
	IF iNoOfEntries > cQueueSize THEN
		bError := TRUE;
	END_IF 
END_IF

// Update input index and find out if queue is full
// bFull := FALSE;
IF((iInputIndex+1) > cQueueSize) THEN
	// Input index has reached end of queue => loop back
	IF(iOutputIndex <> 1 )  THEN
		// Output index is NOT occuping the first index
   		iInputIndex := 1;
  	ELSE
    	// Output index IS occuping the first index => Queue full
		bFull := TRUE;
	 END_IF
ELSE
	// Input index has NOT reach end of queue
	IF((iInputIndex + 1) <> iOutputIndex) THEN
		iInputIndex := iInputIndex + 1;
  	ELSE
		bFull := TRUE;
	END_IF
END_IF

// Update count for number of free entires
iNoOfFree := cQueueSize - iNoOfEntries;
END_METHOD

END_FUNCTION_BLOCK

// ---- POUs/00_BuildingBlocks/Control/FB_RampLimiter.TcPOU
// Ramp function able to ramp in an analog output to an analog input with a given stepsize pr second*)
FUNCTION_BLOCK FB_RampLimiter //Last update: 2016-02-08/ELB
VAR_INPUT
	bEnable				: BOOL;	//Enabling of the ramp. When set FALSE the output is equal to input
	fAI					: REAL;	//Analog input
	fStepSizePrSec		: REAL;	//Size of the step AO is incremented or decremented with pr second
END_VAR
VAR_OUTPUT
	fAO					: REAL; //Analog output
	bError				: BOOL;	//Error
END_VAR
VAR
	fStepSizePrScan		: REAL; //Size of the step AO is incremented or decremented with
	fScanCycleTime_s	: REAL;	//Scan cycle time in s
	fbGetCurTaskIdx 	: GETCURTASKINDEX; //Get current task
END_VAR


// Get current task ID and calculate scan time in sec and step size pr scan
fbGetCurTaskIdx();  
fScanCycleTime_s := UDINT_TO_REAL(_TaskInfo[fbGetCurTaskIdx.index].CycleTime)/10000000; //Find scan time in s
fStepSizePrScan := ABS(fStepSizePrSec*fScanCycleTime_s); //nStepSizePrScanCycle

// Check results. nStepSizePrScan and ScanCycleTime_ms must both be bigger than 0
bERROR := NOT(fStepSizePrScan>0) OR NOT(fScanCycleTime_s>0); 


IF NOT bERROR AND bEnable = TRUE THEN
		
	IF fAO<fAI THEN
		fAO:=fAO+fStepSizePrScan;		//Incremate AO
		IF fAO>fAI THEN 				//AO can not become bigger than AI
			fAO:=fAI;
		END_IF
	END_IF
		
	IF fAO>fAI THEN
		fAO:=fAO-fStepSizePrScan;		//Decremate AO
		IF fAO<fAI THEN 				//AO can not become smaller than AI
			fAO:=fAI; 
		END_IF 	
	END_IF
		
ELSE
	fAO:=fAI;							//If the ramp function is disablet AO=AI no ramp
END_IF

METHOD M_SetOutput : BOOL
VAR_INPUT
	fValue		:REAL;			// Set output value (output jumps to this value)		
END_VAR

fAO := fValue;
END_METHOD

END_FUNCTION_BLOCK

// ---- POUs/00_BuildingBlocks/Control/FB_RangeSupervision.TcPOU
FUNCTION_BLOCK FB_RangeSupervision
VAR_INPUT
	fIn		:REAL;			// Input value
END_VAR
VAR_OUTPUT
	bHiHi	:BOOL;			
	bHi		:BOOL;			
	bLo		:BOOL;			
	bLoLo	:BOOL;				
END_VAR
VAR
	// Inputs from method config
	fHiHi	:REAL;			// Alarm limit high
	fHi		:REAL;			// Warning limit high
	fLo		:REAL;			// Warning limit low
	fLoLo	:REAL;			// Alarm limit low
	
	tHiHi	:TIME;			// Time to activation of high alarm
	tHi		:TIME;			// Time to activation of high warning
	tLo		:TIME;			// Time to activation of low warning
	tLoLo	:TIME;			// Time to activation of low alarm
	
	// Delays
	tonHiHi	:TON;
	tonHi	:TON;
	tonLo	:TON;
	tonLoLo	:TON;
		
	// Before delay is applied for output signal
	bValueHiHi	:BOOL;			
	bValueHi	:BOOL;			
	bValueLo	:BOOL;			
	bValueLoLo	:BOOL;
END_VAR


// Warning limits
FUN_RangeOutside(
	fValue:= fIn, 
	fLimitHigh:= fHi, 
	fLimitLow:= fLo, 
	bHigh=> bValueHi, 
	bLow=> bValueLo);

// Alarm limits
FUN_RangeOutside(
	fValue:= fIn, 
	fLimitHigh:= fHiHi, 
	fLimitLow:= fLoLo, 
	bHigh=> bValueHiHi, 
	bLow=> bValueLoLo);	
	
// Delays
tonHiHi(IN:= bValueHiHi, PT:= tHiHi, Q=> bHiHi);
tonHi(IN:= bValueHi, PT:= tHi, Q=> bHi);
tonLo(IN:= bValueLo, PT:= tLo, Q=> bLo );
tonLoLo(IN:= bValueLoLo, PT:= tLoLo, Q=> bLoLo);

METHOD M_Config : BOOL
VAR_INPUT
	fHiHi	:REAL;			// Alarm limit high
	fHi		:REAL;			// Warning limit high
	fLo		:REAL;			// Warning limit low
	fLoLo	:REAL;			// Alarm limit low
	tHiHi	:TIME;			// Time to activation of high alarm
	tHi		:TIME;			// Time to activation of high warning
	tLo		:TIME;			// Time to activation of low warning
	tLoLo	:TIME;			// Time to activation of low alarm
END_VAR
// Range limits
THIS^.fHiHi := fHiHi;
THIS^.fHi 	:= fHi;
THIS^.fLo 	:= fLo;
THIS^.fLoLo := fLoLo;

// Delay before alarm or warning is set 
THIS^.tHiHi := tHiHi;			
THIS^.tHi 	:= tHi;			
THIS^.tLo 	:= tLo;			
THIS^.tLoLo := tLoLo;
END_METHOD

END_FUNCTION_BLOCK

// ---- POUs/00_BuildingBlocks/Control/FUN_RangeOutside.TcPOU
FUNCTION FUN_RangeOutside : BOOL
VAR_INPUT
	fValue		:REAL;			// Actual value
	fLimitHigh	:REAL;			// High limit for range
	fLimitLow	:REAL;			// Low limit for range
END_VAR
VAR_OUTPUT
	bHigh		:BOOL;			// True if value is greater than rLimitHigh
	bLow		:BOOL;			// True if value is lower than rLimitLow	
END_VAR
VAR
	bOutside	:BOOL;			// True if value is outside of range
END_VAR


// Compare actual value with range
IF fValue < fLimitLow OR fValue > fLimitHigh THEN
	// Outside range
	bOutside := TRUE;
	IF fValue > fLimitHigh THEN
		bHigh := TRUE;
		bLow := FALSE;
	ELSE
		bHigh := FALSE;
		bLow := TRUE;
	END_IF
ELSE
	// Inside of range
	bOutside := FALSE;
END_IF

// Set return value
FUN_RangeOutside := bOutside;

END_FUNCTION

// ---- POUs/00_BuildingBlocks/Control/FB_SignalDead.TcPOU
FUNCTION_BLOCK FB_SignalDead
VAR_INPUT
	fSignal		:REAL;			// Input signal			
	tDelay		:TIME;			// Time from no change in signal to set of output freeze signal
END_VAR
VAR_OUTPUT
	bFreeze		:BOOL;			// Signal is set true if input signal has not changed value within specified time 
END_VAR
VAR
	fSignalOld	:REAL;			// Signal value from previous scan
	tonDelay	:TON;			// Delay from no change in signal to set of output freeze signal
END_VAR


// Check if signal has changed since last scan
//--------------------------------------------------
IF fSignal <> fSignalOld THEN
	// Signal has changed => signal is NOT frozen
	tonDelay(IN:= FALSE);
	bFreeze := FALSE;
ELSE
	// Signal has NOT change => Update timer and evaluate if freeze signal must be set
	tonDelay(IN:= TRUE, PT:=tDelay, Q=> , ET=> );
	IF tonDelay.Q THEN
		bFreeze := TRUE;
	END_IF
END_IF

// Update "old" value
fSignalOld := fSignal;

METHOD M_ResetTime : BOOL
VAR_INPUT
END_VAR
tonDelay(IN:= FALSE);
END_METHOD

END_FUNCTION_BLOCK

// ---- POUs/00_BuildingBlocks/Control/FB_SteadyValue.TcPOU
FUNCTION_BLOCK FB_SteadyValue
VAR_INPUT
	fValue			:REAL;			// Actual value
	fHys			:REAL;			// Hysteresis for acceptance of steady value
	tDelay			:TIME;			// Time where value must be steady
	bLoopBackOn		:BOOL;			// If set true, it is assumed that value will loop back to zero. E.g. at 360 deg.
	fLoopBackLow	:REAL;			// If the input decreases to this value, loop back to fLoopBackHigh occurs
	fLoopBackHigh	:REAL;			// If the input increases to this value, loop back to fLoopBackLow occurs
END_VAR
VAR_OUTPUT
	bSteady			:BOOL;			// True if value is steady (only changing inside hysteresis)
END_VAR
VAR
	bInit			:BOOL:= TRUE;	// True at start of first scan, False otherwise
	fLoopBackLimit	:REAL;
	bLoopBackDetect	:BOOL;
	fValueHigh		:REAL;		
	fValueLow		:REAL;
	fValueOld		:REAL;			// This value is updated to the actual value whenever value is outside of hysteresis
	bDelayOn		:BOOL;
	tonDelay		:TON;			// Timer for steady value
END_VAR

// Initialization
IF bInit THEN
	fValueOld := fValue;
	bDelayOn := FALSE;
	bInit := FALSE;
END_IF

// Determine value +- hysteresis is within reach of loop back
IF bLoopBackOn THEN
	// Loop back is enabled => check if old value is close to loop back points
	IF ((fValueOld + fHys) >= fLoopBackHigh) OR ((fValueOld - fHys) <= fLoopBackLow) THEN
		// Old value is close to loop back.
		IF ((fValueOld + fHys) >= fLoopBackHigh) THEN
			// Old value is close to loop back high
			fLoopBackLimit := fLoopBackLow + ((fValueOld + fHys) - fLoopBackHigh);
			IF ((fValue <= fLoopBackLimit) OR (fValue >= (fValueOld-fHys))) THEN
				// Inside range
				bDelayOn := TRUE;	
			ELSE
				// Outside of range
				bDelayOn := FALSE;
				fValueOld := fValue;
			END_IF
		ELSE
			// Old value is close to loop back low
			fLoopBackLimit := fLoopBackHigh + ((fValueOld - fHys) - fLoopBackLow);
			IF ((fValue >= fLoopBackLimit) OR (fValue <= (fValueOld+fHys))) THEN
				// Inside range
				bDelayOn := TRUE;	
			ELSE
				// Outside of range
				bDelayOn := FALSE;
				fValueOld := fValue;
			END_IF
		END_IF
	ELSE
		// Not close to loop points. Use "normal" limits
		fValueHigh := fValueOld + fHys;
		fValueLow := fValueOld - fHys;
		IF (fValue >= fValueLow) AND (fValue <= fValueHigh) THEN
			// Inside range
			bDelayOn := TRUE;
		ELSE
			// Outside of range
			bDelayOn := FALSE;
			fValueOld := fValue;
		END_IF
	END_IF
ELSE
	// Loop back not enabled. Use "normal" limits
	fValueHigh := fValueOld + fHys;
	fValueLow := fValueOld - fHys;
	IF (fValue >= fValueLow) AND (fValue <= fValueHigh) THEN
		// Inside range
		bDelayOn := TRUE;
	ELSE
		// Outside of range
		bDelayOn := FALSE;
		fValueOld := fValue;
	END_IF	
END_IF

// Set steady value
tonDelay(IN:= bDelayOn, PT:= tDelay, Q=> bSteady, ET=> );

END_FUNCTION_BLOCK

// ---- POUs/00_BuildingBlocks/Control/FUN_InPos.TcPOU
FUNCTION FUN_InPos : BOOL
VAR_INPUT
	rAct_X		:LREAL;			// Actual X-axis position		
	rAct_Y		:LREAL;			// Actual Y-axis position
	rAct_Z		:LREAL;			// Actual Z-axis position
	rSP_X		:LREAL;			// Setpoint X-axis position		
	rSP_Y		:LREAL;			// Setpoint Y-axis position
	rSP_Z		:LREAL;			// Setpoint Z-axis position
	rHys_Mm		:LREAL;			// Hystereis limit for position
	rHys_Deg	:LREAL;			// Hysteresis limit for angle
END_VAR
VAR
	bInPosX		:BOOL;			// True if x-axis position is at setpoint
	bInPosY		:BOOL;			// True if y-axis position is at setpoint
	bInPosZ		:BOOL;			// True if z-axis angle is at setpoint
END_VAR



// Check x-axis position
bInPosX := FUN_InsideHysteresis(rAct:= rAct_X, rSp:= rSP_X, rHys:= rHys_Mm);

// Check y-axis position
bInPosY := FUN_InsideHysteresis(rAct:= rAct_Y, rSp:= rSP_Y, rHys:= rHys_Mm);

// Check z-axis angle
bInPosZ := FALSE;
// Find out if angle is close to switch between 180 and -179.9999 deg.
IF (rSP_Z+rHys_Deg) > 180.0000 OR (rSP_Z-rHys_Deg) < -179.9999 THEN
	// SP is close to switch
	IF rSP_Z > 0 AND rAct_Z >= (rSP_Z-rHys_Deg) AND rAct_Z <= 180.0000 THEN
		// Positive setpoint and actual position inside positve hysteresis area
		bInPosZ := TRUE;
	ELSIF rSP_Z > 0 AND rAct_Z <= (-179.9999 + rHys_Deg -(180-rSP_Z)) AND rAct_Z >= -179.9999 THEN
		// Positive setpoint and actual position inside negative hysteresis area
		bInPosZ := TRUE;
	ELSIF  rSP_Z < 0 AND (rAct_Z <= (rSP_Z+rHys_Deg)) AND rAct_Z >= -179.9999 THEN
		// Negative setpoint and actual position inside negative hysteresis area
		bInPosZ := TRUE;
	ELSIF rSP_Z < 0 AND rAct_Z >= (180- rHys_Deg + (179.9999+rSP_Z)) AND rAct_Z <= 180.0000 THEN
		// Negative setpoint and actual position inside positive hysteresis area
		bInPosZ := TRUE;
	END_IF 
ELSE
	// SP is not close to switch angle
	bInPosZ := FUN_InsideHysteresis(rAct:= rAct_Z, rSp:= rSP_Z, rHys:= rHys_Deg);
END_IF

// Set return value
IF bInPosX AND bInPosY AND bInPosZ THEN
	FUN_InPos := TRUE;
ELSE
	FUN_InPos := FALSE;
END_IF

END_FUNCTION

// ---- POUs/00_BuildingBlocks/Control/FUN_InsideHysteresis.TcPOU
FUNCTION FUN_InsideHysteresis : BOOL
VAR_INPUT
	rAct		:LREAL;			// Actual value
	rSp			:LREAL;			// Setpoint value
	rHys		:LREAL;			// Hysteresis	
END_VAR
VAR
	bInside		:BOOL;			// True if actual value is within setpoint plus minus hysteresis value
END_VAR


// Compare actual value with setpoint and hysteresis limit
IF rAct >= (rSP-rHys) AND rACT <= (rSP+rHys) THEN
	// Inside hysteresis limit
	bInside := TRUE;
ELSE
	// Outside hysteresis limit
	bInside := FALSE;
END_IF

// Set return value
FUN_InsideHysteresis := bInside;

END_FUNCTION

// ---- POUs/00_BuildingBlocks/Control/FUN_InsideHysteresis180pm.TcPOU
FUNCTION FUN_InsideHysteresis180pm : BOOL
VAR_INPUT
	rAct		:REAL;			// [pm 180 deg] Actual value
	rSp			:REAL;			// [pm 180 deg] Setpoint value
	rHys		:REAL;			// [deg] Hysteresis	
END_VAR
VAR
	bInside		:BOOL;			// True if actual value is within setpoint plus minus hysteresis value
END_VAR





// Check z-axis angle
bInside := FALSE;
// Find out if angle is close to switch between 180 and -179.9999 deg.
IF (rSp+rHys) > 180.0000 OR (rSp-rHys) < -179.9999 THEN
	// SP is close to switch
	IF rSp > 0 AND rAct >= (rSp-rHys) AND rAct <= 180.0000 THEN
		// Positive setpoint and actual position inside positve hysteresis area
		bInside := TRUE;
	ELSIF rSp > 0 AND rAct <= (-179.9999 + rHys -(180-rSp)) AND rAct >= -179.9999 THEN
		// Positive setpoint and actual position inside negative hysteresis area
		bInside := TRUE;
	ELSIF  rSp < 0 AND (rAct <= (rSp+rHys)) AND rAct >= -179.9999 THEN
		// Negative setpoint and actual position inside negative hysteresis area
		bInside := TRUE;
	ELSIF rSp < 0 AND rAct >= (180- rHys + (179.9999+rSp)) AND rAct <= 180.0000 THEN
		// Negative setpoint and actual position inside positive hysteresis area
		bInside := TRUE;
	END_IF 
ELSE
	// SP is not close to switch angle
	bInside := FUN_InsideHysteresis(rAct:= rAct, rSp:= rSp, rHys:= rHys);
END_IF

// Set return value
FUN_InsideHysteresis180pm := bInside;

END_FUNCTION

// ---- POUs/00_BuildingBlocks/Control/FUN_InsideHysteresis360.TcPOU
FUNCTION FUN_InsideHysteresis360 : BOOL
VAR_INPUT
	rAct		:REAL;			// Actual value
	rSp			:REAL;			// Setpoint value
	rHys		:REAL;			// Hysteresis	
END_VAR
VAR
	bInside		:BOOL;			// True if actual value is within setpoint plus minus hysteresis value
END_VAR



// Determine if value is close to loop back point at 360 Deg. 
IF (rSp+rHys) > 360.0000 OR (rSp-rHys) < 0.0000 THEN
	// SP is close to switch
	IF (rSp+rHys) > 360.0000 THEN
		// High limit is above 360 deg
		IF (rAct >= (rSp-rHys)) OR (rAct <= (rSp+rHys-360)) THEN
 			bInside := TRUE;
		ELSE
			bInside := FALSE;
		END_IF
	ELSE 
		IF (rAct <= (rSp+rHys)) OR (rAct >= (360+(rSP-rHys))) THEN 
			bInside := TRUE;
		ELSE
			bInside := FALSE;
		END_IF
	END_IF
ELSE
	// SP is not close to 0 or 360 deg.
	bInside := FUN_InsideHysteresis(rAct:= rAct, rSp:= rSp, rHys:= rHys);
END_IF

// Set return value
FUN_InsideHysteresis360 := bInside;

END_FUNCTION

// ---- POUs/00_BuildingBlocks/Control/FUN_RangeInside.TcPOU
FUNCTION FUN_RangeInside : BOOL
VAR_INPUT
	fValue		:LREAL;			// Actual value
	fLimitHigh	:LREAL;			// High limit for range
	fLimitLow	:LREAL;			// Low limit for range
END_VAR
VAR
	bInside		:BOOL;			// True if value is inside range
END_VAR


// Compare actual value with range
IF fValue >= fLimitLow AND fValue <= fLimitHigh THEN
	// Inside range
	bInside := TRUE;
ELSE
	// Outside of range
	bInside := FALSE;
END_IF

// Set return value
FUN_RangeInside := bInside;

END_FUNCTION

// ---- POUs/00_BuildingBlocks/Control/FUN_GetHighLowValue.TcPOU
FUNCTION FUN_GetHighLowValue : UINT
VAR_INPUT
	nValue		:UINT;			// Actual value
END_VAR
VAR_OUTPUT
	nHigh		:UINT;			// True if value is greater than rLimitHigh
	nLow		:UINT;			// True if value is lower than rLimitLow	
END_VAR
VAR
END_VAR

IF nValue > nHigh THEN
	nHigh := nValue;
END_IF

IF nValue < nLow THEN
	nLow := nValue;
END_IF

END_FUNCTION

// ---- POUs/00_BuildingBlocks/Convert/FUN_ConvFourByteToInt32.TcPOU
FUNCTION FUN_ConvFourByteToInt32 : DINT
VAR_INPUT
	nValue1		:BYTE;				// Input Byte no 1
	nValue2		:BYTE;				// Input Byte no 2
	nValue3		:BYTE;				// Input Byte no 3
	nValue4		:BYTE;				// Input Byte no 4
END_VAR
VAR
	uData		:U_Convert_INT32;		// Data variable used for conversion
END_VAR


// Save input bytes in data union
uData.arrByte[1] := nValue1;
uData.arrByte[2] := nValue2;
uData.arrByte[3] := nValue3;
uData.arrByte[4] := nValue4;

// Return value
FUN_ConvFourByteToInt32 := uData.nValue;

END_FUNCTION

// ---- POUs/00_BuildingBlocks/Convert/FUN_ConvFourByteToUdint32.TcPOU
FUNCTION FUN_ConvFourByteToUdint32 : UDINT
VAR_INPUT
	nValue1		:BYTE;				// Input Byte no 1
	nValue2		:BYTE;				// Input Byte no 2
	nValue3		:BYTE;				// Input Byte no 3
	nValue4		:BYTE;				// Input Byte no 4
END_VAR
VAR
	uData		:U_Convert_UDINT32;	// Data variable used for conversion
END_VAR


// Save input bytes in data union
uData.arrByte[1] := nValue1;
uData.arrByte[2] := nValue2;
uData.arrByte[3] := nValue3;
uData.arrByte[4] := nValue4;

// Return value
FUN_ConvFourByteToUdint32 := uData.nValue;

END_FUNCTION

// ---- POUs/00_BuildingBlocks/Convert/FUN_ConvReal32ToFourByte.TcPOU
FUNCTION FUN_ConvReal32ToFourByte : BOOL
VAR_INPUT
	fValue		:REAL;				// Data variable used for conversion
END_VAR
VAR_OUTPUT
	nValue1		:BYTE;				// Output Byte no 1
	nValue2		:BYTE;				// Output Byte no 2
	nValue3		:BYTE;				// OUtput Byte no 3
	nValue4		:BYTE;				// Output Byte no 4
END_VAR
VAR
	uData		:U_Convert_REAL32;	// Data variable used for conversion
END_VAR

// Save input bytes in data union
uData.fValue := fValue;
nValue1 := uData.arrByte[1];
nValue2 := uData.arrByte[2];
nValue3 := uData.arrByte[3];
nValue4 := uData.arrByte[4];

END_FUNCTION

// ---- POUs/00_BuildingBlocks/Convert/FUN_ConvTwoByteToInt16.TcPOU
FUNCTION FUN_ConvTwoByteToInt16 : INT
VAR_INPUT
	nValue1		:BYTE;				// Input Byte no 1
	nValue2		:BYTE;				// Input Byte no 2
END_VAR
VAR
	uData		:U_Convert_INT16;		// Data variable used for conversion
END_VAR


// Save input bytes in data union
uData.arrByte[1] := nValue1;
uData.arrByte[2] := nValue2;

// Return value
FUN_ConvTwoByteToInt16 := uData.nValue;

END_FUNCTION

// ---- POUs/00_BuildingBlocks/Convert/FUN_ConvOneByteToUint8.TcPOU
FUNCTION FUN_ConvOneByteToUint8 : UINT
VAR_INPUT
	nValue1		:BYTE;				// Input Byte no 1

END_VAR
VAR
	uData		:U_Convert_UINT8;		// Data variable used for conversion
END_VAR

// Save input bytes in data union
uData.nBYTE := nValue1;


// Return value
FUN_ConvOneByteToUInt8 := uData.nValue;

END_FUNCTION

// ---- POUs/00_BuildingBlocks/EtherCAT/FB_EK1101_Check.TcPOU
//********************************************************************************
// FB_EK1101_Check
// -------------------------------------------------------------------------------
//  This FB checks the status for an EtherCAT coupler
//
//  V2.00.01, HHL, nState is moved to input (Due to project structure)
//	V2.00.00, HHL, Baseline Unknown, 24/08-2016
//********************************************************************************
FUNCTION_BLOCK FB_EK1101_Check
VAR_INPUT
	nState					:UINT;			// ID switch number input
END_VAR
VAR_OUTPUT
	bSlaveError				:BOOL;			// On if slave has error
	sSlaveState				:STRING(80);	// State description
END_VAR
VAR
	iAlive					:INT;			// FB alive counter	

END_VAR


// Alive counter.
iAlive:=iAlive+1;

// Initialize slate state
sSlaveState:='';

// State
IF nState > 0 THEN
	
	bSlaveError:=TRUE;
	
	IF nState = 1 THEN
		sSlaveState:=' Slave in "INIT" state';
	END_IF
	
	IF nState = 1 THEN
		sSlaveState:=' Slave in "INIT" state';
	END_IF
	
	IF nState = 2 THEN
		sSlaveState:=' Slave in "PREOP" state';
	END_IF
	
	IF nState = 3 THEN
		sSlaveState:=' Slave in "BOOT" state';
	END_IF
	
	IF nState = 4 THEN
		sSlaveState:=' Slave in "SAFEOP" state';
	END_IF
	
	IF nState = 8 THEN
		sSlaveState:=' Slave in "OPERATIONEL" state';
		bSlaveError := FALSE;
	END_IF
	
	IF nState > 8 THEN
		sSlaveState:=' Slave in "ERROR" state and NOT operationel';
	END_IF
ELSE
	sSlaveState:= 'No connection to coupler.';
	bSlaveError:= TRUE;
END_IF

//***********************************  State info:
//
(*
0x___1 = Slave in 'INIT' state
0x___2 = Slave in 'PREOP' state
0x___3 = Slave in 'BOOT' state
0x___4 = Slave in 'SAFEOP' state
0x___8 = Slave in 'OP' state
0x001_ = Slave signals error
0x002_ = Invalid vendorId, productCode... read
0x004_ = Initialization error occurred
0x008_ = Slave disabled
0x010_ = Slave not present
0x020_ = Slave signals link error
0x040_ = Slave signals missing link
0x080_ = Slave signals unexpected link
0x100_ = Communication port A
0x200_ = Communication port B
0x400_ = Communication port C
0x800_ = Communication port D
*)

END_FUNCTION_BLOCK

// ---- POUs/00_BuildingBlocks/EtherCAT/FB_HardwareCheck.TcPOU
FUNCTION_BLOCK FB_HardwareCheck
VAR_INPUT
	nState					: UINT; // Status input from terminal
	bAlarmIn				: BOOL; // If this is active, dont check alarm status for next terminal
END_VAR
VAR_OUTPUT
	bAlarm					: BOOL; // Active alarm on terminal
END_VAR
VAR
	nOperationState			: UINT := 8; // Terminal is in normal operation
END_VAR

// Only check for alarms if no alarms is present in last terminal, and the machine is in IO mode for hardware
IF GVL_Hmi.stHw.stSta.eIfSource = E_System_IfSources.IO THEN
	IF bAlarmIn = FALSE THEN
		// Check if terminal status == 8 (Operation)
		IF nState <> nOperationState THEN
			bAlarm := TRUE;
		ELSE
			bAlarm := FALSE;
		END_IF
	END_IF
	
ELSE
	// Reset the alarm output if was true when sources mode was changed
	bAlarm := FALSE;
END_IF

END_FUNCTION_BLOCK

// ---- POUs/00_BuildingBlocks/File/FB_FileHandler.TcPOU
FUNCTION_BLOCK FB_FileHandler
VAR_INPUT
	bReset				:BOOL;						// Reset active error on rising edge
END_VAR

VAR_OUTPUT
	bReady				:BOOL;						// True when FileHandler is ready for new cmd
	bError				:BOOL;						// True if error occured during operation
END_VAR

VAR
	// State variables
	bInit				:BOOL:=TRUE;				// True in start of first scan, otherwise false
	bEntry				:BOOL;						// True in first scan when entering a new state
	eStep				:E_FileHandler_State;		// Active state
	eStepPrevious			:E_FileHandler_State;		// State in previous scan	
	bLocked				:BOOL;						// True if state machine is locked
	bCmdReadFile		:BOOL;						// Command for read file
	bCmdWriteFile		:BOOL;						// Command for write lines to file
	bCmdCopyFile		:BOOL;						// Command for copying file
	bCmdDelFile			:BOOL;						// Command for deleting file
	bUseMountAndCopy	:BOOL;						// Signal for use of mount and copy batch script instead of just copy
	
	// FB's for file handling
	fbFileOpen			:FB_FileOpen;				// Opens a file
	fbFileRead			:FB_FileRead;				// Reads content of file and stores in byte array from file
	fbFileWrite			:FB_FileWrite;				// Writes lines from array of strings to file
	fbFileClose			:FB_FileClose;				// Closes a file

	// Variables for file handling
	sFileNameAndPath	:STRING(255);					// File name and path
	uiFileHandle		:UINT;						// File handle
	arrFileData			:ARRAY[0..cNoOfBytesMax] OF BYTE; // Array with all data from file
	pFileLines			:POINTER TO ARRAY[1..GVL_Constants.cFileReadNoOfLines] OF STRING(80); // Pointer to array with one entry for each line in file 
	pNoOfLines			:POINTER TO UDINT;			// Number of lines in file

	// Write
	iWriteNoOfLines		:INT;						// Number of lines to be written 
	pWriteLines			:POINTER TO ARRAY[1..GVL_Constants.cFileWriteNoOfLines] OF STRING(500); // Pointer to array of lines that must be written to a file
	sWriteLine			:STRING(500);				// String to be written to file
	iWriteLineIndex		:INT;						// Index for number of written lines
	iWriteLineLength	:UDINT;						// Length of line
	
	// Read
	udiActiveByte		:UDINT;						// Active byte for processing
	udiStartByte		:UDINT;						// Start byte during processing
	iActiveLine			:UDINT;						// Active line for processing of data to strings
	iScanLineCount		:UDINT;						// Counts the number of lines that has been read in one scan
	iLineReturnCount	:INT;						// Counts the number of scans used to read the file

	// Copy
	fbBatchCopyExe		:NT_StartProcess;			// FB that starts the batch file which copies file from servers
	sCopyFileName		:STRING(80);				// File to be copied
	sCopyFromFolder		:STRING(175);				// Folder where file is copied from
	sCopyToFolder		:STRING(175);				// Folder where file is copied to
	sCopyCmdLine		:STRING(380);				// Command line 
	sCopyDirName		:STRING(175) := 'C:\Epex2\Control\Batch\';
	sCopyPathString		:STRING(255) := 'C:\Epex2\Control\Batch\CopyFile.bat';
	
	// Del
	fbBatchDelExe		:NT_StartProcess;			// FB that starts the batch file which copies file from servers
	sDelFileName		:STRING(80);				// File to be copied
	sDelFromFolder		:STRING(175);				// Folder where file is copied from
	sDelCmdLine			:STRING(380);				// Command line
	sDelDirName			:STRING(175) := 'C:\Epex2\Control\Batch\';
	sDelPathString		:STRING(255) := 'C:\Epex2\Control\Batch\DeleteFile.bat';
	
	// Error
	bErrFileOpen		:BOOL;						// Error when file was opened
	bErrFileRead		:BOOL;						// Error when file was read	
	bErrFileWrite		:BOOL;						// Error when file was written
	bErrFileClose		:BOOL;						// Error when file was closed
	bErrFileCopy		:BOOL;						// Error when file was copied
	bErrFileDel			:BOOL;						// Error when file was deleted
END_VAR
VAR CONSTANT
	cNoOfBytesMax		:UDINT := 2000000;			// Maximum number of bytes in file
	cLinesInOneScanMax	:UDINT := 150;				// Maximum number of lines read in one scan
END_VAR

// Initialization
//-----------------------------------------
IF bInit THEN
	eStepPrevious := eStep;
	bInit := FALSE;
END_IF



// Set ready flag
//-----------------------------------------
bReady := (eStep = E_FileHandler_State.eIdle) AND NOT bLocked;



// Call file FB's
//-----------------------------------------
A_UpdateFileFBs();

	
	
// State machine for file handler
//-----------------------------------------
// Set entry flag
IF eStep <> eStepPrevious THEN
	bEntry := TRUE;
ELSE
	bEntry := FALSE;
END_IF
eStepPrevious := eStep;


CASE eStep OF

// Initialization
E_FileHandler_State.eReset:
	// Entry
	IF bEntry THEN
		;
	END_IF
	eStep := E_FileHandler_State.eIdle;
	
// Idle
E_FileHandler_State.eIdle:
	// Entry
	IF bEntry THEN
		// Reset any errors
		bError := FALSE;
		bErrFileOpen := FALSE;
		bErrFileRead := FALSE;
		bErrFileWrite := FALSE;
		bErrFileClose := FALSE;
		bErrFileCopy := FALSE;	
	END_IF
	
	// Check for new commands
	IF bCmdReadFile OR bCmdWriteFile THEN
		// Reset lock
		bLocked := FALSE;
		eStep := E_FileHandler_State.eOpenFilePre;
	ELSIF bCmdCopyFile THEN
		// Copy file
		bLocked := FALSE;
		eStep := E_FileHandler_State.eCopyFilePre;
	ELSIF bCmdDelFile THEN
		// Delete file
		bLocked := FALSE;
		eStep := E_FileHandler_State.eDelFilePre;
	END_IF
	
	
// Open file Pre
E_FileHandler_State.eOpenFilePre:
	// Entry
	IF bEntry THEN
		fbFileOpen(bExecute:=FALSE);
		fbFileOpen.tTimeout := T#3S;
		fbFileOpen.sPathName := sFileNameAndPath;
		IF bCmdReadFile THEN
			fbFileOpen.nMode := FOPEN_MODEREAD;		// Read only mode
		ELSIF bCmdWriteFile THEN
			fbFileOpen.nMode := FOPEN_MODEAPPEND;	
		END_IF
		fbFileOpen.tTimeout := T#3S;
	END_IF
	
	// Start execute of file open and wait for busy flag
	fbFileOpen.bExecute := TRUE;
	IF fbFileOpen.bBusy THEN 
		// Open is in progress go and wait for done
		eStep := E_FileHandler_State.eOpenFilePeri;
	END_IF
	
	
	
// Open file Peri
E_FileHandler_State.eOpenFilePeri:
	// Entry
	IF bEntry THEN
		;
	END_IF
	
	// Wait for done
	IF NOT fbFileOpen.bBusy AND NOT fbFileOpen.bError THEN
		uiFileHandle := fbFileOpen.hFile;
		IF bCmdReadFile THEN
			eStep := E_FileHandler_State.eReadFilePre;
		ELSIF bCmdWriteFile THEN
			eStep := E_FileHandler_State.eWriteFilePre;
		END_IF
	ELSIF fbFileOpen.bError THEN
		bErrFileOpen := TRUE;
 		eStep := E_FileHandler_State.eErrEntry;
	END_IF



// Read file Pre
E_FileHandler_State.eReadFilePre:
	// Entry
	IF bEntry THEN
		fbFileRead(bExecute:=FALSE);
		fbFileRead.hFile := uiFileHandle;
		fbFileRead.pReadBuff := ADR(arrFileData);
		fbFileRead.cbReadLen := cNoOfBytesMax;
	END_IF
	
	// Start file reading		
	fbFileRead.bExecute:= TRUE;
	IF fbFileRead.bBusy  THEN
		// File reading has begun, Go and wait for it to finish
		eStep := E_FileHandler_State.eReadFilePeri;
	END_IF

	
	
// Read file Peri
E_FileHandler_State.eReadFilePeri:
	// Entry
	IF bEntry THEN
		;
	END_IF
	
	// Wait for done
	IF NOT fbFileRead.bBusy AND NOT fbFileRead.bError THEN
		// File was succesfulle read
		eStep := E_FileHandler_State.eCloseFilePre;
	ELSIF fbFileRead.bError THEN
		// Error occured
		bErrFileRead := TRUE;
 		eStep := E_FileHandler_State.eErrEntry;
	END_IF

	
	
// Write file Pre
E_FileHandler_State.eWriteFilePre:
	// Entry
	IF bEntry THEN
		fbFileWrite(bExecute:=FALSE);
		fbFileWrite.hFile := uiFileHandle;
		iWriteLineIndex := 1;
	END_IF	
	eStep := E_FileHandler_State.eWriteFileSetLine;

	
	
// Write file, Set line
E_FileHandler_State.eWriteFileSetLine:	
	IF bEntry THEN
		sWriteLine := '';
		sWriteLine := pWriteLines^[iWriteLineIndex];
		iWriteLineLength := LEN2(pSTRING:= ADR(sWriteLine));
		fbFileWrite.pWriteBuff := ADR(sWriteLine);
		fbFileWrite.cbWriteLen := iWriteLineLength;
		fbFileWrite.bExecute:= TRUE;	
	END_IF	
	eStep := E_FileHandler_State.eWriteFilePeri;
	

	
// Write file Peri
E_FileHandler_State.eWriteFilePeri:
	// Entry
	IF bEntry THEN
		;
	END_IF	
	
	// Wait untill write operation is finished
	IF NOT fbFileWrite.bBusy AND NOT fbFileWrite.bError THEN		
		IF iWriteLineIndex < iWriteNoOfLines THEN 
			// More lines must be written. Go back and write next line	   
			eStep := E_FileHandler_State.eWriteFileSetLine;
			iWriteLineIndex := iWriteLineIndex + 1;
		ELSE
			// All lines have been written => close file 
			eStep := E_FileHandler_State.eCloseFilePre;
		END_IF;
		fbFileWrite(bExecute:=FALSE);	
	ELSIF fbFileWrite.bError THEN
		bErrFileWrite := TRUE;
		eStep := E_FileHandler_State.eErrEntry;
	END_IF

	
	
// Close file Pre
E_FileHandler_State.eCloseFilePre:
	// Entry
	IF bEntry THEN
		fbFileClose(bExecute:=FALSE);
		fbFileClose.hFile := uiFileHandle;
	END_IF
	
	// Start file closing			
	fbFileClose.bExecute:= TRUE;
	IF fbFileClose.bBusy THEN
		// Close has begun, Go and wait for close to end	
		eStep := E_FileHandler_State.eCloseFilePeri;
	END_IF

	
	
// Close file Peri
E_FileHandler_State.eCloseFilePeri:
	// Entry
	IF bEntry THEN
		;
	END_IF
	
	// Wait for done
	IF NOT fbFileClose.bBusy AND NOT fbFileClose.bError THEN
		// File was succesfulle closed
		IF bCmdReadFile THEN
			eStep := E_FileHandler_State.eProcessFile;
		ELSIF bCmdWriteFile THEN
			bCmdWriteFile := FALSE;
			eStep := E_FileHandler_State.eIdle;
		END_IF
	ELSIF fbFileClose.bError THEN
		bErrFileClose := TRUE;
 		eStep := E_FileHandler_State.eErrEntry;
	END_IF

	
	
// Process file content
E_FileHandler_State.eProcessFile:	
		// Entry
	IF bEntry THEN
		pNoOfLines^ := 0;
		iActiveLine := 1;
		pFileLines^[1] := ''; 
		iScanLineCount := 0;
		udiStartByte := 0;
		iLineReturnCount := 1;
	END_IF
	
	// Process data
	FOR udiActiveByte := udiStartByte TO fbFileRead.cbRead DO
		IF  F_ToCHR(arrFileData[udiActiveByte]) = '$N'  THEN;
			// New line
			iActiveLine := iActiveLine +1;
			iScanLineCount := iScanLineCount +1;			
			pFileLines^[iActiveLine] := '';
			IF iScanLineCount >= cLinesInOneScanMax THEN
				iScanLineCount := 0;
				udiStartByte := udiActiveByte + 1;
				iLineReturnCount := iLineReturnCount + 1;
				RETURN;
			END_IF
		ELSIF NOT (F_ToCHR(arrFileData[udiActiveByte]) = '$R') THEN
			// Return => store data up untill this point as a line
			pFileLines^[iActiveLine] := CONCAT(pFileLines^[iActiveLine], F_ToCHR(arrFileData[udiActiveByte]));
		END_IF
	END_FOR

	// Check if all data has been processed
	IF udiActiveByte >= fbFileRead.cbRead THEN
		pNoOfLines^ := iActiveLine-1;
		bCmdReadFile := FALSE;
		eStep := E_FileHandler_State.eIdle;
	END_IF

	
// Copy file pre	
E_FileHandler_State.eCopyFilePre:
	// Entry
	IF bEntry THEN
		
		// Check for backslah at end of string for "from" folder 
		IF RIGHT(sCopyFromFolder,1) <> '\' THEN 
			sCopyFromFolder := CONCAT(sCopyFromFolder,'\');
		END_IF
	
		// Check for backslah at end of string for "to" folder
		IF RIGHT(sCopyToFolder,1) <> '\' THEN 
			sCopyToFolder := CONCAT(sCopyToFolder,'\');
		END_IF
		
		// Check if copy to folder is on local or external drive
		IF (MID(sCopyToFolder, 1, 1) <> 'c') AND (MID(sCopyToFolder, 1, 1) <> 'C') THEN
			// Server (switch server drive letter to 'x')
			sCopyToFolder := REPLACE(sCopyToFolder,'x', 1, 1);
			bUseMountAndCopy := TRUE;
		ELSE
			bUseMountAndCopy := FALSE;
		END_IF
		
		// Create command line
		sCopyFromFolder := CONCAT('"',sCopyFromFolder);
		sCopyFileName := CONCAT(sCopyFileName,'"');
		sCopyCmdLine := CONCAT(sCopyFromFolder, sCopyFileName); 
		sCopyCmdLine := CONCAT(sCopyCmdLine, ' ');
		sCopyCmdLine := CONCAT(sCopyCmdLine, sCopyToFolder);
		
		// Check if copy is from local or external drive
		IF ((MID(sCopyCmdLine, 1, 2) = 'c') OR (MID(sCopyCmdLine, 1, 2) = 'C')) AND NOT bUseMountAndCopy THEN
			// From local to local drive
			// Initialize fb that starts copy function
			fbBatchCopyExe(START:= FALSE); 
			fbBatchCopyExe.PATHSTR:= sCopyPathString; 
			fbBatchCopyExe.DIRNAME:= sCopyDirName; 
			fbBatchCopyExe.COMNDLINE:= sCopyCmdLine; 
			fbBatchCopyExe.TMOUT:= T#5S;
		ELSIF ((MID(sCopyCmdLine, 1, 2) = 'c') OR (MID(sCopyCmdLine, 1, 2) = 'C')) AND bUseMountAndCopy THEN
			// To server from local drive
			// Initialize fb that starts copy function
			fbBatchCopyExe(START:= FALSE); 
			fbBatchCopyExe.PATHSTR:= 'C:\Epex2\Control\Batch\MountAndCopyFile.bat'; 
			fbBatchCopyExe.DIRNAME:= sCopyDirName; 
			fbBatchCopyExe.COMNDLINE:= sCopyCmdLine; 
			fbBatchCopyExe.TMOUT:= T#5S;
		ELSE
			// From server to local drive (switch server drive letter to 'x')
			sCopyCmdLine := REPLACE(sCopyCmdLine,'x', 1, 2);
			// Initialize fb that starts copy function
			fbBatchCopyExe(START:= FALSE); 
			fbBatchCopyExe.PATHSTR:= 'C:\Epex2\Control\Batch\MountAndCopyFile.bat'; 
			fbBatchCopyExe.DIRNAME:= sCopyDirName; 
			fbBatchCopyExe.COMNDLINE:= sCopyCmdLine; 
			fbBatchCopyExe.TMOUT:= T#5S;
		END_IF
	END_IF
	
	// Start batch file for copy		
	fbBatchCopyExe.START:= TRUE;
	IF fbBatchCopyExe.BUSY THEN
		fbBatchCopyExe.START:= FALSE; 
		// Open is in progress go and wait for done
		eStep := E_FileHandler_State.eCopyFilePeri;
	END_IF

	
	
// Copy file peri
 E_FileHandler_State.eCopyFilePeri:
 	// Entry
	IF bEntry THEN
		;
	END_IF
 
	// Wait for done
	IF NOT fbBatchCopyExe.BUSY AND NOT fbBatchCopyExe.ERR  THEN
		// Copy process was succesfulle started
		bCmdCopyFile := FALSE; 
		eStep := E_FileHandler_State.eIdle;
	ELSIF fbBatchCopyExe.ERR THEN
		// Error occured
		bCmdCopyFile := FALSE;
		bErrFileCopy := TRUE;
 		eStep := E_FileHandler_State.eErrEntry;
	END_IF
	
	
	
// Delete file pre	
E_FileHandler_State.eDelFilePre:
	// Entry
	IF bEntry THEN
		// Create command line
		sDelFromFolder := CONCAT('"',sDelFromFolder);
		sDelFileName := CONCAT(sDelFileName,'"');
		sDelCmdLine := CONCAT(sDelFromFolder, sDelFileName); 
		// Initialize fb that starts delete function
		fbBatchDelExe(START:= FALSE); 
		fbBatchDelExe.PATHSTR:= sDelPathString; 
		fbBatchDelExe.DIRNAME:= sDelDirName; 
		fbBatchDelExe.COMNDLINE:= sDelCmdLine; 
		fbBatchDelExe.TMOUT:= T#5S;
	END_IF
	
	// Start batch file for delete		
	fbBatchDelExe.START:= TRUE;
	IF fbBatchDelExe.BUSY THEN
		fbBatchDelExe.START:= FALSE; 
		// Open is in progress go and wait for done
		eStep := E_FileHandler_State.eDelFilePeri;
	END_IF

	
	
// Delete file peri
 E_FileHandler_State.eDelFilePeri:
 	// Entry
	IF bEntry THEN
		;
	END_IF
 
	// Wait for done
	IF NOT fbBatchDelExe.BUSY AND NOT fbBatchDelExe.ERR  THEN
		// Del process was succesfulle started
		bCmdDelFile := FALSE; 
		eStep := E_FileHandler_State.eIdle;
	ELSIF fbBatchDelExe.ERR THEN
		// Error occured
		bCmdDelFile := FALSE;
		bErrFileDel := TRUE;
 		eStep := E_FileHandler_State.eErrEntry;
	END_IF	
	
	
	
	

// Error states
// Error entry state
E_FileHandler_State.eErrEntry:
	// Entry
	IF bEntry THEN
		bError := TRUE;
	END_IF
		
	// Identify error
	IF bErrFileOpen THEN
		eStep := E_FileHandler_State.eErrOpen;
	ELSIF bErrFileRead THEN
		eStep := E_FileHandler_State.eErrRead;
	ELSIF bErrFileWrite THEN
		eStep := E_FileHandler_State.eErrWrite;
	ELSIF bErrFileClose THEN
		eStep := E_FileHandler_State.eErrClose;
	ELSIF bErrFileCopy THEN
		eStep := E_FileHandler_State.eErrCopy;
	ELSIF bErrFileDel THEN
		eStep := E_FileHandler_State.eErrDel;		
	END_IF
	
	
	
// Error open file
E_FileHandler_State.eErrOpen:
	// Entry
	IF bEntry THEN
		bCmdReadFile := FALSE;
	END_IF

	// Reset => Go back and wait for new command
	IF bReset THEN
		eStep := E_FileHandler_State.eIdle;
	END_IF
	

// Error read file
E_FileHandler_State.eErrRead:
	// Entry
	IF bEntry THEN
		bCmdReadFile := FALSE;
	END_IF
	
	// Reset => Go back and wait for new command
	IF bReset THEN
		fbFileRead(bExecute := FALSE);
		eStep := E_FileHandler_State.eIdle;
	END_IF
	


// Error write file
E_FileHandler_State.eErrWrite:
	// Entry
	IF bEntry THEN
		bCmdWriteFile := FALSE;
	END_IF
		
	// Reset => Go back and wait for new command
	IF bReset THEN
		fbFileWrite(bExecute:= FALSE);
		eStep := E_FileHandler_State.eIdle;
	END_IF
	
	
	
// Error close file
E_FileHandler_State.eErrClose:
	// Entry
	IF bEntry THEN
		;
	END_IF
		
	// Reset => Go back and wait for new command
	IF bReset THEN
		fbFileClose(bExecute:= FALSE);
		eStep := E_FileHandler_State.eIdle;
	END_IF

	
	
// Error copy file
E_FileHandler_State.eErrCopy:
	// Entry
	IF bEntry THEN
		;
	END_IF
		
	// Reset => Go back and wait for new command
	IF bReset THEN
		fbBatchCopyExe(START:= FALSE);
		eStep := E_FileHandler_State.eIdle;
	END_IF

	

// Error copy file
E_FileHandler_State.eErrDel:
	// Entry
	IF bEntry THEN
		;
	END_IF
		
	// Reset => Go back and wait for new command
	IF bReset THEN
		fbBatchDelExe(START:= FALSE);
		eStep := E_FileHandler_State.eIdle;
	END_IF
END_CASE

ACTION A_UpdateFileFBs:
fbFileOpen(
	sNetId:= , 
	sPathName:= , 
	nMode:= , 
	ePath:= , 
	bExecute:= , 
	tTimeout:= , 
	bBusy=> , 
	bError=> , 
	nErrId=> , 
	hFile=> );
	
fbFileRead(
	sNetId:= , 
	hFile:= , 
	pReadBuff:= , 
	cbReadLen:= , 
	bExecute:= , 
	tTimeout:= , 
	bBusy=> , 
	bError=> , 
	nErrId=> , 
	cbRead=> , 
	bEOF=> );
	
fbFileWrite(
	sNetId:= , 
	hFile:= , 
	pWriteBuff:= , 
	cbWriteLen:= , 
	bExecute:= , 
	tTimeout:= , 
	bBusy=> , 
	bError=> , 
	nErrId=> , 
	cbWrite=> );	
	
fbFileClose(
	sNetId:= , 
	hFile:= , 
	bExecute:= , 
	tTimeout:= , 
	bBusy=> , 
	bError=> , 
	nErrId=> );
	
fbBatchCopyExe(
	NETID:= , 
	PATHSTR:= , 
	DIRNAME:= , 
	COMNDLINE:= , 
	START:= , 
	TMOUT:= , 
	BUSY=> , 
	ERR=> , 
	ERRID=> );	
	
fbBatchDelExe(
	NETID:= , 
	PATHSTR:= , 
	DIRNAME:= , 
	COMNDLINE:= , 
	START:= , 
	TMOUT:= , 
	BUSY=> , 
	ERR=> , 
	ERRID=> );
END_ACTION

METHOD M_CopyFile : BOOL
VAR_INPUT
	sFileName			:STRING(80);					// Filename
	sFilePathFrom		:STRING(175);					// File path
	sFilePathTo			:STRING(175);					// Local folder where file must be copied to
END_VAR

// Set execute flag if it is a valid command
IF eStep = E_FileHandler_State.eIdle AND NOT bLocked THEN
	// State machine is idle => Copy is a valid command
	sCopyFileName := sFileName;
	sCopyFromFolder := sFilePathFrom;
	sCopyToFolder := sFilePathTo;	
	bLocked := TRUE;
	bReady	:= FALSE;
	bCmdCopyFile := TRUE;
END_IF

// Return boolean value for execution accept.
IF bCmdCopyFile THEN
	M_CopyFile := TRUE;
ELSE
	M_CopyFile := FALSE;
END_IF
END_METHOD

METHOD M_DeleteFile : BOOL
VAR_INPUT
	sFileName			:STRING(80);					// Filename
	sFileFolder			:STRING(175);					// File path
END_VAR

// Set execute flag if it is a valid command
IF eStep = E_FileHandler_State.eIdle AND NOT bLocked THEN
	// State machine is idle => Delete is a valid command
	sDelFileName := sFileName;
	sDelFromFolder := sFileFolder;
	bLocked := TRUE;
	bReady	:= FALSE;
	bCmdDelFile := TRUE;
END_IF

// Return boolean value for execution accept.
IF bCmdDelFile THEN
	M_DeleteFile := TRUE;
ELSE
	M_DeleteFile := FALSE;
END_IF
END_METHOD

METHOD M_ReadFile : BOOL
VAR_INPUT
	sFileName			:STRING(80);					// Filename
	sFilePath			:STRING(175);					// File path
	pArrLines			:POINTER TO ARRAY[1..GVL_Constants.cFileReadNoOfLines] OF STRING(80); // Pointer ot array with one entry for each line in file
	pLinesInFile		:POINTER TO UDINT;			// Variable where no of lines is stored 
END_VAR
// Set execute flag if it is a valid command
IF eStep = E_FileHandler_State.eIdle AND NOT bLocked THEN
	// State machine is idle => Read is a valid command
	sFileNameAndPath := CONCAT(sFilePath,sFileName);
	pFileLines := pArrLines;
	pNoOfLines := pLinesInFile;
	bLocked := TRUE;
	bReady	:= FALSE;
	bCmdReadFile := TRUE;
END_IF

// Return boolean value for execution accept.
IF bCmdReadFile THEN
	M_ReadFile := TRUE;
ELSE
	M_ReadFile := FALSE;
END_IF
END_METHOD

METHOD M_WriteFile : BOOL
VAR_INPUT
	sFileName			:STRING(80);					// Filename
	sFilePath			:STRING(175);					// File path
	iLinesToWrite		:INT;						// Number of lines to written from array of strings				
	pArrLines			:POINTER TO ARRAY[1..GVL_Constants.cFileWriteNoOfLines] OF STRING(500); // Pointer ot array with one entry for each line in file
END_VAR
// Set execute flag if it is a valid command
IF eStep = E_FileHandler_State.eIdle AND NOT bLocked AND iLinesToWrite > 0 THEN
	// State machine is idle => Read is a valid command
	sFileNameAndPath := CONCAT(sFilePath,sFileName);
	iWriteNoOfLines	:= iLinesToWrite;
	pWriteLines := pArrLines;
	bLocked := TRUE;
	bReady	:= FALSE;
	bCmdWriteFile := TRUE;
END_IF

// Return boolean value for execution accept.
IF bCmdWriteFile THEN
	M_WriteFile := TRUE;
ELSE
	M_WriteFile := FALSE;
END_IF
END_METHOD

END_FUNCTION_BLOCK

// ---- POUs/00_BuildingBlocks/Modbus/FB_ModbusRtuMaster.TcPOU
// FB_ModbusMaster
//------------------------------------------------------
// This FB must be called in a 2 ms task and in every scan
// Test with Danfoss FC301 shows that up to approximately 46 registers can be read pr. sec.
// Test was done with baud 115200. 
// V 1.1, Updated so that Modbus master continues to next unit if an error occurs.  
// V 1.0, Baseline. Developed december 2021 
FUNCTION_BLOCK FB_ModbusRtuMaster
VAR_INPUT
	pUnit					:POINTER TO ARRAY[1..cNoOfUnitsMax] OF ST_Modbus_Unit;
	nNoOfUnits				:INT;			// Number of modbus units. Maximum value is 20.					
	nNoOfParam				:INT;			// Number of modbus parameters to be read from unit. Maximum value is determined by ST_Modbus_Unit. 
END_VAR
VAR_OUTPUT
	bBusy					:BOOL;			// True while command is beeing executed
	bError					:BOOL;			// True if an error occured during execution of a command
	nErrorUnit				:INT;			// First unit where error was detected in communication
END_VAR
VAR
	// Commands
	bCmdCyclicRead			:BOOL;			// Command for cyclic reading of parameter registers
	bCmdStop				:BOOL;			// Command for stop
	bCmdReset				:BOOL;			// Command for reset of active errors
	
	// General	
	bInit					:BOOL := TRUE;	// True at the start of false scan, false otherwise
	nReadCount				:INT;			// Counts the number of succesfull read operations
	nValueTempInt16			:INT;			// Value used in conversion from byte data to actual data value
	nValueTempInt32			:DINT;			// Value used in conversion from byte data to actual data value
	
